(* CODESYS project xlh_ha_00_02.project
   Author: Pascal Helfenstein
   Title: xlh_ha
   Company: xemax ag

Project tree, tasks and I/O mapping:
  xlh_base : CODESYS Control for Raspberry Pi 64 SL, CODESYS, order no. 2302000009, version 4.20.0.0
    application app
      libraries: Standard, 3.5.22.0 (System); StringUtils, 3.5.22.0 (System); VisuDialogs, * (System); Web Socket Client SL, 1.12.0.0 (CODESYS); Net Base Services, * (3S - Smart Software Solutions GmbH); MQTT Client SL, 1.13.0.0 (CODESYS); Util, 3.5.22.0 (System); String Functions, * (CODESYS); SysTimeRtc, * (System); SysTime, 3.5.17.0 (System); CmpIecTask, * (System); Memory, 3.5.17.0 (3S - Smart Software Solutions GmbH)
      task MainTask (cyclic, interval t#20ms, priority 1) calls LOCAL_TIME_AND_TIME_ZONE, TASK_INFO, io, MAIN
      task VISU_TASK (cyclic, interval 100 ms, priority 31) calls VisuElems.Visu_Prg
      program MAIN [ST]
      IoT/
        DEVICES/
          function block _000_FB_VISU_BASE [ST]
          function block _200_FB_DEVICE_SHELLY_BASE [ST]: statusUpdate, startup, newMessage
          function block _202_FB_DEVICE_SHELLY_1PM_TEMP [ST]: newMessage
          interface IDevice
          interface IDeviceZigbee2Mqtt
          interface IDeviceShelly
          function block _201_FB_DEVICE_SHELLY_1PM_PLUG [ST]: publisher, newMessage
          function block _300_FB_DEVICE_Z2M_BASE [ST]: statusUpdate, startup, newMessage
          VISU/
            visualisation VISU_FB_DEVICE_SHELLY_RELAIS
            visualisation VISU_FB_DEVICE_SHELLY_RELAIS_TEMP
            visualisation _310_VISU_FB_DEVICE_Z2M_POWER_SWITCH
            visualisation _311_VISU_FB_DEVICE_Z2M_POWER_SWITCH_IKEAL_INSPELING
            visualisation _312_VISU_FB_DEVICE_Z2M_POWER_LAMP
            visualisation _341_VISU_FB_DEVICE_Z2M_BATTERY_SONOFF_TEMP_HUM
          function block _100_FB_DEVICE [ST]: subscriber, publisher, startup, popFifoPublish, newMessage, statusUpdate, pushFifoPublish
          interface IVisu
          function block _311_FB_DEVICE_Z2M_POWER_SWITCH_IKEA_INSPELING [ST]: newMessage
          function block _312_FB_DEVICE_Z2M_POWER_LAMP [ST]: newMessage, publisher
          function block _310_FB_DEVICE_Z2M_POWER_SWITCH [ST]: statusUpdate, startup, newMessage, publisher
          function block _341_FB_DEVICE_Z2M_BATTERY_SONOFF_TEMP_HUM [ST]: newMessage
          function block _340_FB_DEVICE_Z2M_BATTERY [ST]: newMessage
          function block _342_FB_DEVICE_Z2M_BATTERY_AQARA_SWITCH_H1 [ST]: newMessage
          function block _314_FB_DEVICE_Z2M_SHELLY_EM [ST]: newMessage
          function block _343_FB_DEVICE_Z2M_BATTERY_HUE_SWITCH_DIMMER [ST]: newMessage
          function block _344_FB_DEVICE_Z2M_BATTERY_HUE_MOTION [ST]: newMessage
          function block _345_FB_DEVICE_Z2M_BATTERY_HUE_WALL_SWITCH [ST]: newMessage
          function block _313_FB_DEVICE_Z2M_SHELLY_1PM [ST]: newMessage
        MQTT_Client/
          function TERMINATE_STRING [ST]
          function block FB_MQTT_CLIENT [ST]: pMqttClient, setClientIdNr
          function GET_VALUE_FROM_MSG [ST]
          function GET_REAL_FROM_VALUE [ST]
          function GET_BOOL_FROM_VALUE [ST]
          function GET_INT_FROM_VALUE [ST]
          function GET_STRING_FROM_VALUE [ST]
          function GET_LREAL_FROM_VALUE [ST]
          function GET_BOOL_FROM_VALUE_ON_OFF [ST]
        global variables GC
        program TASK_INFO [ST]
        program LOCAL_TIME_AND_TIME_ZONE [ST]
        FUNCTIONS/
          function block FB_IMPULSE_SWITCH [ST]
      visualisation VISUALIZATION
      io/
        program io [ST]
      program LOGIC [CFC]
    SoftMotion General Axis Pool
    GPIOs_A_B : GPIOs B+/Pi2, CODESYS, version 4.20.0.0
        unmapped channels: digital inputs (GPIO0..GPIO31), digital outputs (GPIO0..GPIO31)
    Onewire
    Camera device
      <Empty>
    SPI
    I²C
  libraries: VisuSymbols, 4.5.0.0 (System)
  text list GlobalTextList
  5ce3da45-db07-42e7-a21c-a00fff4ed8f6|C:\Users\a.werner\Documents\background.jpg
*)

// xlh_base/app/IoT/GC
// =============================================================================
// GC — Global constants (qualified-only)
// -----------------------------------------------------------------------------
// Collects the string sizes used project-wide for MQTT topics and message
// buffers. Changes affect the memory footprint of every device FB.
// =============================================================================
{attribute 'qualified_only'}
VAR_GLOBAL CONSTANT
    STRING_SIZE_TOPIC      : INT := 1024;   // Maximum size of an MQTT topic ((W)STRING length)
    STRING_SIZE_MESSAGE_TX : INT := 1024;   // Maximum size of a transmit message
    STRING_SIZE_MESSAGE_RX : INT := 2048;   // Maximum size of a receive message
END_VAR

// xlh_base/app/IoT/LOCAL_TIME_AND_TIME_ZONE
// =============================================================================
// LOCAL_TIME_AND_TIME_ZONE
// -----------------------------------------------------------------------------
// Provides the current UTC and CET/CEST time and their components
// (year, month, day, hour, ..., weekday, leap year) as program outputs.
//
// Uses the Util library for the time-zone conversion between UTC (RTC)
// and Central European Time (daylight-saving switchover on the last
// Sunday of March/October respectively).
//
// Usage: time-of-day controls (e.g. _344 motion sensor active window).
// =============================================================================
PROGRAM LOCAL_TIME_AND_TIME_ZONE
VAR_OUTPUT
    stUTC_Timestamp      : SysTime;         // RTC timestamp UTC
    stCTE_Timestamp      : SysTime;         // CET/CEST timestamp
    stJoinedTimestamp    : SysTime;         // CET components joined back into a UTC timestamp
    stCombinedTimestamp  : SysTime;         // datDate + todTime combined
    uiYear               : YEAR;            // 1970..2106
    uiMonth              : MONTH;
    uiDay                : DAY;
    uiHour               : UINT;
    uiMinute             : UINT;
    uiSecond             : UINT;
    uiMilliseconds       : MILLISECOND;
    eWeekday             : WEEKDAY;
    datDate              : DATE;
    todTime              : TIME_OF_DAY;
    eError               : Util.ERROR;
    xLeapYear            : BOOL;
END_VAR
VAR CONSTANT
    /// Coordinated Universal Time
    gc_tzTimeZoneUTC : TimeZone := (asgPeriod := [(sName := 'UTC')]);

    /// Central European Time / Central European Summer Time with switchover rules.
    gc_tzTimeZoneCET : TimeZone := (
        iBias := 60 (* T#1M => minutes *),
        asgPeriod := [
            ( (* Summer time -> standard time: last Sunday of October, 03:00 local *)
                sName  := 'CET',
                dtDate := (uiMonth := 10, eWeekday := WEEKDAY.SUNDAY, uiDay := 5, uiHour := 3)
            ),
            ( (* Standard time -> summer time: last Sunday of March, 02:00 local *)
                sName  := 'CEST',
                dtDate := (uiMonth := 3,  eWeekday := WEEKDAY.SUNDAY, uiDay := 5, uiHour := 2),
                iBias  := 60 (* T#1M => minutes *)
            )
        ]
    );
END_VAR

// 1) Read the RTC UTC timestamp.
SysTimeRtcHighResGet(pTimestamp := stUTC_Timestamp);

// 2) UTC -> CET/CEST according to the configured TimeZone.
stCTE_Timestamp := Util.LocalDateTime(tzTimeZone := gc_tzTimeZoneCET,
                                      uliDateTime := stUTC_Timestamp,
                                      eErrorID    => eError);

// 3) Split the CET timestamp into its individual components.
eError := Util.SplitDateTime(uliDateTime    := stCTE_Timestamp,
                             uiYear         => uiYear,
                             uiMonth        => uiMonth,
                             uiDay          => uiDay,
                             uiHour         => uiHour,
                             uiMinute       => uiMinute,
                             uiSecond       => uiSecond,
                             uiMilliseconds => uiMilliseconds,
                             eWeekday       => eWeekday);

// 4) Join the components back into a UTC timestamp (diagnostics).
stJoinedTimestamp := Util.JoinDateTime(uiYear         := uiYear,
                                       uiMonth        := uiMonth,
                                       uiDay          := uiDay,
                                       uiHour         := uiHour,
                                       uiMinute       := uiMinute,
                                       uiSecond       := uiSecond,
                                       uiMilliseconds := uiMilliseconds);

// 5) Derive the IEC-typed parts (datDate, todTime).
Util.SeparateDateTime(uliDateTime := stCTE_Timestamp,
                      eWeekDay    => eWeekDay,
                      datDate     => datDate,
                      todTime     => todTime);

// 6) Reconstruct a timestamp from datDate + todTime.
stCombinedTimestamp := Util.CombineDateTime(datDate  := datDate,
                                            todTime  := todTime,
                                            eErrorID => eError);

// 7) Calculate the weekday from the date (verification).
eWeekday := Util.DayOfWeek(datDate := datDate, eErrorID => eError);

// 8) Leap-year flag.
xLeapYear := Util.IsLeapYear(uiYear := uiYear, eErrorID => eError);

END_PROGRAM

// xlh_base/app/IoT/TASK_INFO
// =============================================================================
// TASK_INFO
// -----------------------------------------------------------------------------
// Reads the key figures of the current task (interval, jitter, effective
// cycle time) at runtime via the CmpIecTask library and makes them available
// to all POUs through program outputs.
//
// Usage in the device FBs: integration of energy via fCycleTime, periodic
// status queries via fCycleTime-based second counters.
//
// Sources:
//   https://content.helpme-codesys.com/en/libs/CmpIecTask/Current/index.html
//   https://forge.codesys.com/forge/talk/Engineering/thread/b7e9b2b353/
//   https://medium.com/@sean.gongz/...how-to-get-current-task-actual-cycle-time-in-codesys
// =============================================================================
PROGRAM TASK_INFO
VAR
    Result            : CmpIecTask.RTS_IEC_RESULT;
    hCurrentTask      : CmpIecTask.RTS_IEC_HANDLE;
    pCurrentTaskInfo  : POINTER TO Task_Info2;
    stCurrentTaskInfo : Task_Info2;
END_VAR
VAR_OUTPUT
    fCycleTime              : LREAL;    // Effective cycle time in seconds (interval + jitter)
    fInterval               : LREAL;    // Configured task interval (us)
    fCycleTimeUs            : LREAL;    // Effective cycle time in microseconds
    fJitterUs               : LREAL;    // Current jitter (us)
    fJitterOffsetInterwalUs : LREAL;    // Interval + jitter (us)
END_VAR

// Get the current task handle and dereference the info structure.
hCurrentTask      := IecTaskGetCurrent(pResult := ADR(Result));
pCurrentTaskInfo  := IecTaskGetInfo3(hIecTask := hCurrentTask, pResult := ADR(Result));
stCurrentTaskInfo := pCurrentTaskInfo^;

// Prepare the results.
fCycleTimeUs            := TO_LREAL(TO_DINT(stCurrentTaskInfo.dwInterval) + stCurrentTaskInfo.iJitter);
fInterval               := TO_LREAL(stCurrentTaskInfo.dwInterval);
fJitterUs               := TO_LREAL(stCurrentTaskInfo.iJitter);
fJitterOffsetInterwalUs := fInterval + fJitterUs;
fCycleTime              := fCycleTimeUs / 1000000.0;

END_PROGRAM

// xlh_base/app/io/io
// =============================================================================
// io
// -----------------------------------------------------------------------------
// Central device program: instantiates all devices connected via
// Zigbee2MQTT/Shelly (as VAR_INPUT so they can be parameterized via the
// visualization / online), binds them to shared FB_MQTT_CLIENT instances
// and calls them cyclically.
//
// Architecture:
//   - Devices are not assigned directly to one MQTT client but are managed
//     through a pointer array (_aIoClients).
//   - Several FB_MQTT_CLIENT instances (_afbMqttClient) are used so that
//     the MQTT library is not overloaded by too many parallel subscribes.
//     iNR_OF_IO_TO_ONE_MQTT_CLIENT devices are bundled per MQTT client.
//   - The initial configuration (pointer binding, topics) is done once in
//     the startup block.
// =============================================================================
PROGRAM io
VAR_INPUT
    // Zigbee wireless switches / sensors (battery devices)
    fbSwitch1       : _343_FB_DEVICE_Z2M_BATTERY_HUE_SWITCH_DIMMER := (bEnable:=TRUE, sMqttTopicBase:='switch_1', sLabel:='');
    fbSwitch2       : _345_FB_DEVICE_Z2M_BATTERY_HUE_WALL_SWITCH   := (bEnable:=TRUE, sMqttTopicBase:='switch_2', sLabel:='');
    fbTempHumSensor : _341_FB_DEVICE_Z2M_BATTERY_SONOFF_TEMP_HUM   := (bEnable:=TRUE, sMqttTopicBase:='temp_hum_sensor', sLabel:='');
    fbMotionSensor: _344_FB_DEVICE_Z2M_BATTERY_HUE_MOTION       := (bEnable:=TRUE, sMqttTopicBase:='motion_sensor', sLabel:='');

    // Zigbee switch actuators / lamps / energy meters
    fbLamp1   : _312_FB_DEVICE_Z2M_POWER_LAMP                       := (bEnable:=TRUE, sMqttTopicBase:='lamp_1',  sLabel:='');
    fbLamp2   : _312_FB_DEVICE_Z2M_POWER_LAMP                       := (bEnable:=TRUE, sMqttTopicBase:='lamp_2',  sLabel:='');
    fbPlug1   : _310_FB_DEVICE_Z2M_POWER_SWITCH                     := (bEnable:=TRUE, sMqttTopicBase:='plug_1',  sLabel:='');
    fbPlug2   : _311_FB_DEVICE_Z2M_POWER_SWITCH_IKEA_INSPELING      := (bEnable:=TRUE, sMqttTopicBase:='plug_2',  sLabel:='');
    fbShelly1 : _313_FB_DEVICE_Z2M_SHELLY_1PM                       := (bEnable:=TRUE, sMqttTopicBase:='shelly_1', sLabel:='');
    fbShelly2 : _314_FB_DEVICE_Z2M_SHELLY_EM                        := (bEnable:=TRUE, sMqttTopicBase:='shelly_2', sLabel:='');
END_VAR
VAR CONSTANT
    iNR_OF_IO_CLIENTS            : INT := 100; // Maximum number of devices in the pointer array
    iNR_OF_MQTT_CLIENTS          : INT :=  20; // Number of MQTT clients (connections to the broker)
    iNR_OF_IO_TO_ONE_MQTT_CLIENT : INT :=   5; // Devices per MQTT client
END_VAR
VAR
    _bStartup     : BOOL := TRUE;                                                     // One-time initialization
    _aIoClients   : ARRAY[0..(iNR_OF_IO_CLIENTS   - 1)] OF POINTER TO _100_FB_DEVICE; // Device pointer array
    _afbMqttClient: ARRAY[0..(iNR_OF_MQTT_CLIENTS - 1)] OF FB_MQTT_CLIENT;            // Distributed MQTT clients
    _iI           : INT;
    _iN           : INT;
END_VAR

// =============================================================================
// One-time initialization
// -----------------------------------------------------------------------------
// 1. Register the devices in the pointer array (the order determines the
//    assignment to the MQTT clients).
// 2. Set the ClientId per MQTT client (xlh_base_ha_io_<n>).
// 3. Bind the devices to their MQTT client pointer and call startup().
// 4. Enable the MQTT clients (bEnable := TRUE).
// =============================================================================
IF _bStartup THEN
    _bStartup := FALSE;

    // (1) Register the devices.
    _iI := 0;
    _aIoClients[_iI] := ADR(fbSwitch1);       _iI := _iI + 1;
    _aIoClients[_iI] := ADR(fbSwitch2);       _iI := _iI + 1;
    _aIoClients[_iI] := ADR(fbTempHumSensor); _iI := _iI + 1;
    _aIoClients[_iI] := ADR(fbMotionSensor);  _iI := _iI + 1;

    _aIoClients[_iI] := ADR(fbLamp1);         _iI := _iI + 1;
    _aIoClients[_iI] := ADR(fbLamp2);         _iI := _iI + 1;
    _aIoClients[_iI] := ADR(fbPlug1);         _iI := _iI + 1;
    _aIoClients[_iI] := ADR(fbPlug2);         _iI := _iI + 1;
    _aIoClients[_iI] := ADR(fbShelly1);       _iI := _iI + 1;
    _aIoClients[_iI] := ADR(fbShelly2);       _iI := _iI + 1;

    // (2) Set unique client ids.
    FOR _iI := 0 TO (iNR_OF_MQTT_CLIENTS - 1) BY 1 DO
        _afbMqttClient[_iI].setClientIdNr(sClientId := 'xlh_base_ha_io_', iNr := _iI);
    END_FOR

    // (3) Bind the devices to the MQTT clients and initialize them.
    FOR _iI := 0 TO (iNR_OF_IO_CLIENTS - 1) BY 1 DO
        IF _aIoClients[_iI] > 16#0 THEN
            _iN := _iI / iNR_OF_IO_TO_ONE_MQTT_CLIENT;
            _aIoClients[_iI]^.pMqttClient := ADR(_afbMqttClient[_iN]);
            _aIoClients[_iI]^.startup();
        END_IF
    END_FOR

    // (4) Enable the MQTT clients.
    FOR _iI := 0 TO (iNR_OF_MQTT_CLIENTS - 1) BY 1 DO
        _afbMqttClient[_iI].bEnable := TRUE;
    END_FOR
END_IF

// =============================================================================
// Cyclic calls
// =============================================================================
// MQTT clients first -> required so the subscribers/publishers of the
// devices see an up-to-date connection state.
FOR _iI := 0 TO (iNR_OF_MQTT_CLIENTS - 1) BY 1 DO
    _afbMqttClient[_iI]();
END_FOR

// Call the devices.
FOR _iI := 0 TO (iNR_OF_IO_CLIENTS - 1) BY 1 DO
    IF _aIoClients[_iI] > 16#0 THEN
        _aIoClients[_iI]^();
    END_IF
END_FOR

END_PROGRAM

// xlh_base/app/IoT/MQTT_Client/FB_MQTT_CLIENT
// =============================================================================
// FB_MQTT_CLIENT
// -----------------------------------------------------------------------------
// Wrapper around the IoTCommonLib MQTT.MQTTClient. Provides a simplified
// interface (Enable / Hostname / ClientId) and returns the connection and
// error status flags.
//
// Properties / methods:
//   - pMqttClient    : Property GET, returns a pointer to the internal MQTT
//                      client (used by device FBs to bind their own
//                      subscribe/publish blocks to the client).
//   - setClientIdNr  : Helper method to create a unique client id by
//                      appending a sequential number.
// =============================================================================
FUNCTION_BLOCK FB_MQTT_CLIENT
VAR_INPUT
    bEnable   : BOOL;                       // TRUE = activate the connection
    sHostname : STRING(255) := 'localhost'; // Hostname of the MQTT broker
    sClientId : STRING(255) := 'xLH_mqtt_codesys'; // Unique client id
END_VAR
VAR_OUTPUT
    bConnected  : BOOL;                     // TRUE = connected to the broker
    bError      : BOOL;                     // TRUE = connection/protocol error
    fbMqttClient: MQTT.MQTTClient := (
        uiPort             := 1883,
        eMQTTVersion       := MQTT.MQTT_VERSION.V3_1_1,
        eCommunicationMode := MQTT.COMMUNICATION_MODE.TCP); // Internal client (referenced by pMqttClient)
END_VAR

// Control the MQTT client: while the error flag is active, xEnable is
// automatically reset so the IoTCommon library can reset internally.
fbMqttClient.xEnable   := bEnable AND NOT fbMqttClient.xError;
fbMqttClient.sClientId := sClientId;
fbMqttClient(sHostname := sHostname);

// Status outputs.
bConnected := fbMqttClient.xConnectedToBroker;
bError     := fbMqttClient.xError;

// =============================================================================
// PROPERTY pMqttClient (GET)
// -----------------------------------------------------------------------------
// Returns a pointer to the internal MQTT client so that device FBs can
// couple their MQTT.MQTTSubscribe / MQTT.MQTTPublish instances to the same
// connection.
// =============================================================================
PROPERTY pMqttClient : POINTER TO FB_MQTT_CLIENT
GET
pMqttClient := ADR(THIS^.fbMqttClient);
END_GET
END_PROPERTY

// =============================================================================
// METHOD setClientIdNr
// -----------------------------------------------------------------------------
// Sets the client id by appending a sequential number to a base name.
// Used by the io program to create a unique id per MQTT client instance
// ('xlh_base_ha_io_0', '..._1', ...).
// =============================================================================
METHOD setClientIdNr : BOOL
VAR_INPUT
    sClientId : STRING(255) := 'xLH_mqtt_codesys'; // Base id
    iNr       : INT;                                // Number to append
END_VAR
VAR
    sNumber : STRING(255);
END_VAR
sNumber := TO_STRING(iNr);
THIS^.sClientId := CONCAT(sClientId, sNumber);
END_METHOD

END_FUNCTION_BLOCK

// xlh_base/app/IoT/DEVICES/_343_FB_DEVICE_Z2M_BATTERY_HUE_SWITCH_DIMMER
// =============================================================================
// _343_FB_DEVICE_Z2M_BATTERY_HUE_SWITCH_DIMMER
// -----------------------------------------------------------------------------
// Philips Hue Dimmer Switch (4 buttons: On / Off / Up / Down) with
// press / hold / release actions per button.
// Device link: https://www.zigbee2mqtt.io/devices/929002398602.html
//
// Behavior of the boolean outputs:
//   - Pulses: set for EXACTLY ONE PLC cycle when an action is received,
//     reset again in the following cycle.
// =============================================================================
FUNCTION_BLOCK _343_FB_DEVICE_Z2M_BATTERY_HUE_SWITCH_DIMMER EXTENDS _340_FB_DEVICE_Z2M_BATTERY
VAR_OUTPUT
    sAction          : STRING(255);   // Last reported action (diagnostics)

    // ON button
    bOnPress         : BOOL;
    bOnPressRelease  : BOOL;
    bOnHold          : BOOL;
    bOnHoldRelease   : BOOL;

    // OFF button
    bOffPress        : BOOL;
    bOffPressRelease : BOOL;
    bOffHold         : BOOL;
    bOffHoldRelease  : BOOL;

    // UP button
    bUpPress         : BOOL;
    bUpPressRelease  : BOOL;
    bUpHold          : BOOL;
    bUpHoldRelease   : BOOL;

    // DOWN button
    bDownPress       : BOOL;
    bDownPressRelease: BOOL;
    bDownHold        : BOOL;
    bDownHoldRelease : BOOL;
END_VAR
VAR
    _bNewAction : BOOL;
END_VAR

SUPER^();

IF _bNewAction THEN
    _bNewAction := FALSE;

    bOnPress          := sAction = 'on_press';
    bOnPressRelease   := sAction = 'on_press_release';
    bOnHold           := sAction = 'on_hold';
    bOnHoldRelease    := sAction = 'on_hold_release';

    bOffPress         := sAction = 'off_press';
    bOffPressRelease  := sAction = 'off_press_release';
    bOffHold          := sAction = 'off_hold';
    bOffHoldRelease   := sAction = 'off_hold_release';

    bUpPress          := sAction = 'up_press';
    bUpPressRelease   := sAction = 'up_press_release';
    bUpHold           := sAction = 'up_hold';
    bUpHoldRelease    := sAction = 'up_hold_release';

    bDownPress        := sAction = 'down_press';
    bDownPressRelease := sAction = 'down_press_release';
    bDownHold         := sAction = 'down_hold';
    bDownHoldRelease  := sAction = 'down_hold_release';
ELSE
    bOnPress          := FALSE;
    bOnPressRelease   := FALSE;
    bOnHold           := FALSE;
    bOnHoldRelease    := FALSE;

    bOffPress         := FALSE;
    bOffPressRelease  := FALSE;
    bOffHold          := FALSE;
    bOffHoldRelease   := FALSE;

    bUpPress          := FALSE;
    bUpPressRelease   := FALSE;
    bUpHold           := FALSE;
    bUpHoldRelease    := FALSE;

    bDownPress        := FALSE;
    bDownPressRelease := FALSE;
    bDownHold         := FALSE;
    bDownHoldRelease  := FALSE;
END_IF

// =============================================================================
// METHOD newMessage
// -----------------------------------------------------------------------------
// Reads the action from the event topic and triggers the pulse logic in
// the next cycle.
// =============================================================================
METHOD newMessage : BOOL
SUPER^.newMessage();
IF _fbMqttSubscriber.wsLastTopic = _wsMqttTopicEvent THEN
    sAction := GET_STRING_FROM_VALUE(sAction, GET_VALUE_FROM_MSG('action', ADR(_sSubscribedMessage)));
    THIS^._bNewAction := TRUE;
END_IF
END_METHOD

END_FUNCTION_BLOCK

// xlh_base/app/IoT/DEVICES/_340_FB_DEVICE_Z2M_BATTERY
// =============================================================================
// _340_FB_DEVICE_Z2M_BATTERY
// -----------------------------------------------------------------------------
// Base FB for battery-powered Zigbee devices. Reads the battery level
// (battery, 0..100%) from the Z2M event topic.
//
// Derived by sensors (_341, _344) and push buttons/switches (_342, _343,
// _345).
// =============================================================================
FUNCTION_BLOCK _340_FB_DEVICE_Z2M_BATTERY EXTENDS _300_FB_DEVICE_Z2M_BASE
VAR_OUTPUT
    iBattery : INT := -1;       // Battery level 0..100% (-1 = unknown)
END_VAR

SUPER^();

// =============================================================================
// METHOD newMessage
// -----------------------------------------------------------------------------
// Reads the battery level from the Z2M event topic.
// =============================================================================
METHOD newMessage : BOOL
SUPER^.newMessage();
IF _fbMqttSubscriber.wsLastTopic = _wsMqttTopicEvent THEN
    iBattery := GET_INT_FROM_VALUE(iBattery, GET_VALUE_FROM_MSG('battery', ADR(_sSubscribedMessage)));
END_IF
END_METHOD

END_FUNCTION_BLOCK

// xlh_base/app/IoT/DEVICES/_300_FB_DEVICE_Z2M_BASE
// =============================================================================
// _300_FB_DEVICE_Z2M_BASE
// -----------------------------------------------------------------------------
// Base FB for Zigbee2MQTT devices. Provides the standard Z2M topics and
// parses the common 'linkquality' field.
//
// Standard topic schema (Zigbee2MQTT):
//   zigbee2mqtt/<base>          (subscribe filter via wildcard ".../#")
//   zigbee2mqtt/<base>          -> event topic (status pushes from the device)
//   zigbee2mqtt/<base>/set      -> publish: action to the device
//   zigbee2mqtt/<base>/get      -> publish: trigger a status query
//
// Example:
//   Set output
//     zigbee2mqtt/plug_1/set    {"state": "OFF"} | {"state": "ON"}
//   Status query
//     zigbee2mqtt/plug_1/get    {"state":""}
// =============================================================================
FUNCTION_BLOCK _300_FB_DEVICE_Z2M_BASE EXTENDS _100_FB_DEVICE IMPLEMENTS IDeviceZigbee2Mqtt
VAR_INPUT
    sMqttTopicZigbee2Mqtt : STRING(255) := 'zigbee2mqtt';   // Z2M prefix (usually 'zigbee2mqtt')
END_VAR
VAR_OUTPUT
    iLinkquality : INT := -1;       // Zigbee link quality (-1 = unknown)
END_VAR
VAR
    _wsMqttTopicZigbee2Mqtt : WSTRING(GC.STRING_SIZE_TOPIC); // sMqttTopicZigbee2Mqtt as WSTRING
    _wsMqttTopicEvent       : WSTRING(GC.STRING_SIZE_TOPIC); // zigbee2mqtt/<base>
    _wsMqttTopicSet         : WSTRING(GC.STRING_SIZE_TOPIC); // zigbee2mqtt/<base>/set
    _wsMqttTopicGet         : WSTRING(GC.STRING_SIZE_TOPIC); // zigbee2mqtt/<base>/get
END_VAR

SUPER^();

// =============================================================================
// METHOD statusUpdate
// -----------------------------------------------------------------------------
// Hook (no own code) — overridden by derived FBs.
// =============================================================================
METHOD statusUpdate : BOOL
SUPER^.statusUpdate();
END_METHOD

// =============================================================================
// METHOD startup
// -----------------------------------------------------------------------------
// Builds the subscribe filter and all Z2M-specific topic strings.
// =============================================================================
METHOD startup : BOOL
SUPER^.startup();
THIS^._wsMqttTopicZigbee2Mqtt := STRING_TO_WSTRING(sMqttTopicZigbee2Mqtt);

// Subscribe filter: zigbee2mqtt/<base>/#
_wsSubcribedTopicFilter := "";
Stu.StrConcatW(pstFrom:=ADR(THIS^._wsMqttTopicZigbee2Mqtt), pstTo:=ADR(_wsSubcribedTopicFilter), iBufferSize:=GC.STRING_SIZE_TOPIC);
Stu.StrConcatW(pstFrom:=ADR("/"),                          pstTo:=ADR(_wsSubcribedTopicFilter), iBufferSize:=GC.STRING_SIZE_TOPIC);
Stu.StrConcatW(pstFrom:=ADR(THIS^._wsMqttTopicBase),       pstTo:=ADR(_wsSubcribedTopicFilter), iBufferSize:=GC.STRING_SIZE_TOPIC);
Stu.StrConcatW(pstFrom:=ADR("/#"),                         pstTo:=ADR(_wsSubcribedTopicFilter), iBufferSize:=GC.STRING_SIZE_TOPIC);

// Event topic: zigbee2mqtt/<base>
_wsMqttTopicEvent := "";
Stu.StrConcatW(pstFrom:=ADR(THIS^._wsMqttTopicZigbee2Mqtt), pstTo:=ADR(_wsMqttTopicEvent), iBufferSize:=GC.STRING_SIZE_TOPIC);
Stu.StrConcatW(pstFrom:=ADR("/"),                          pstTo:=ADR(_wsMqttTopicEvent), iBufferSize:=GC.STRING_SIZE_TOPIC);
Stu.StrConcatW(pstFrom:=ADR(THIS^._wsMqttTopicBase),       pstTo:=ADR(_wsMqttTopicEvent), iBufferSize:=GC.STRING_SIZE_TOPIC);

// Set topic: zigbee2mqtt/<base>/set
_wsMqttTopicSet := "";
Stu.StrConcatW(pstFrom:=ADR(_wsMqttTopicEvent), pstTo:=ADR(_wsMqttTopicSet), iBufferSize:=GC.STRING_SIZE_TOPIC);
Stu.StrConcatW(pstFrom:=ADR("/set"),            pstTo:=ADR(_wsMqttTopicSet), iBufferSize:=GC.STRING_SIZE_TOPIC);

// Get topic: zigbee2mqtt/<base>/get
_wsMqttTopicGet := "";
Stu.StrConcatW(pstFrom:=ADR(_wsMqttTopicEvent), pstTo:=ADR(_wsMqttTopicGet), iBufferSize:=GC.STRING_SIZE_TOPIC);
Stu.StrConcatW(pstFrom:=ADR("/get"),            pstTo:=ADR(_wsMqttTopicGet), iBufferSize:=GC.STRING_SIZE_TOPIC);
END_METHOD

// =============================================================================
// METHOD newMessage
// -----------------------------------------------------------------------------
// Reads the link quality (available for all Z2M devices) from the event
// topic.
// =============================================================================
METHOD newMessage : BOOL
SUPER^.newMessage();
IF _fbMqttSubscriber.wsLastTopic = _wsMqttTopicEvent THEN
    iLinkquality := GET_INT_FROM_VALUE(iLinkquality, GET_VALUE_FROM_MSG('linkquality', ADR(_sSubscribedMessage)));
END_IF
END_METHOD

END_FUNCTION_BLOCK

// xlh_base/app/IoT/DEVICES/_100_FB_DEVICE
// =============================================================================
// _100_FB_DEVICE
// -----------------------------------------------------------------------------
// Generic MQTT device base class. Connects one MQTT subscriber and one MQTT
// publisher instance to an externally referenced FB_MQTT_CLIENT and provides
// a publish queue (LIFO).
//
// Usage:
//   1. Externally assign pMqttClient (pointer to FB_MQTT_CLIENT) and
//      sMqttTopicBase in the calling program.
//   2. Call the method startup() once for commissioning (the topic filters
//      are built).
//   3. bEnable := TRUE -> the subscriber subscribes to sMqttTopicBase + '/#'
//      and calls newMessage() for every message.
//
// Extension in derived FBs:
//   - newMessage()    : Parse the message and update the outputs.
//   - publisher()     : Enqueue MQTT messages via pushFifoPublish().
//   - statusUpdate()  : Called once on every subscribe re-/connect
//                       (e.g. to send active status queries).
//
// Publish queue:
//   The methods push/popFifoPublish implement a LIFO with a fixed depth of
//   _iFIFO_SIZE. An internal cycle-delay counter prevents several publishes
//   from following each other without a pause (relieves the broker and the
//   MQTT library).
// =============================================================================
FUNCTION_BLOCK _100_FB_DEVICE EXTENDS _000_FB_VISU_BASE IMPLEMENTS IDevice
VAR_INPUT
    bEnable        : BOOL;                          // TRUE -> subscriber/publisher active
    sMqttTopicBase : STRING(255);                   // Base topic of the device (without wildcard)
    pMqttClient    : POINTER TO FB_MQTT_CLIENT;     // Pointer to the shared MQTT client
END_VAR
VAR
    // ---- Topic strings (caches) -----------------------------------------------
    _wsMqttTopicBase         : WSTRING(GC.STRING_SIZE_TOPIC); // sMqttTopicBase as WSTRING
    _wsSubcribedTopicFilter  : WSTRING(GC.STRING_SIZE_TOPIC); // _wsMqttTopicBase + '/#'

    // ---- Connection triggers and watchdogs ------------------------------------
    _fbRtMqttClientConnected : R_TRIG;                // Rising edge:  MQTT connection established
    _fbFtMqttClientConnected : F_TRIG;                // Falling edge: MQTT connection lost
    _fbRtMqttSubscriberActive: R_TRIG;                // Subscriber became active (-> statusUpdate)
    _fbFtMqttSubscriberActive: F_TRIG;
    _fbRtError               : R_TRIG;                // Error edge of the MQTT client
    _fbTonConnect            : TON;                   // Reconnect delay (subscribe enable)
    _fbTonDisconnect         : TON;                   // Watchdog (subscribe disable when stale)

    // ---- Subscriber -----------------------------------------------------------
    _fbMqttSubscriber : MQTT.MQTTSubscribe;
    _sSubscribedMessage : STRING(GC.STRING_SIZE_MESSAGE_RX);

    // ---- Publisher (current slot) ---------------------------------------------
    _fbMqttPublisher : MQTT.MQTTPublish;
    _wsPublishTopic  : WSTRING(GC.STRING_SIZE_TOPIC);
    _sPublishMessage : STRING(GC.STRING_SIZE_MESSAGE_TX);

    // ---- Publisher queue (LIFO) -----------------------------------------------
    _iFifoPos             : INT;       // Current fill level
    _iFifoPosMax          : INT;       // Maximum value (watermark) for diagnostics
    _iFifoPopCycleCounter : INT;       // Cycle delay between pop operations
    _awsPublishTopic   : ARRAY[0..(_iFIFO_SIZE - 1)] OF WSTRING(GC.STRING_SIZE_TOPIC);
    _asPublishMessage  : ARRAY[0..(_iFIFO_SIZE - 1)] OF STRING(GC.STRING_SIZE_MESSAGE_TX);

    // ---- Diagnostics ----------------------------------------------------------
    _todMessageUpdate : TIME_OF_DAY;   // Time of day of the last received message
END_VAR
VAR CONSTANT
    _iFIFO_SIZE          : INT := 30; // Depth of the publish queue
    _iFIFO_DELAY_COUNTER : INT := 5;  // Cycles of pause between two publish pop operations
END_VAR

THIS^.subscriber();
THIS^.publisher();

// =============================================================================
// METHOD subscriber
// -----------------------------------------------------------------------------
// Manages the life cycle of the MQTT subscriber and calls newMessage() for
// new messages and statusUpdate() on (re-)activation.
//
// Logic:
//   - The subscriber is activated when the connection is established and
//     deactivated on disconnect / error.
//   - Watchdog _fbTonDisconnect (3s): if the subscriber is enabled but not
//     busy, it is briefly disabled to reset the library.
//   - After _fbTonConnect (500ms) the subscriber is activated again.
// =============================================================================
METHOD subscriber : BOOL
THIS^._fbRtMqttClientConnected(CLK := THIS^.pMqttClient^.bConnected);
THIS^._fbFtMqttClientConnected(CLK := THIS^.pMqttClient^.bConnected);
THIS^._fbRtError              (CLK := THIS^.pMqttClient^.bError);

// Activate the subscriber on connect, deactivate it on error/disconnect.
IF THIS^._fbRtMqttClientConnected.Q THEN
    THIS^._fbMqttSubscriber.xEnable := TRUE;
END_IF
IF THIS^._fbRtError.Q OR THIS^._fbFtMqttClientConnected.Q THEN
    THIS^._fbMqttSubscriber.xEnable := FALSE;
END_IF

// Watchdog: stalled subscriber -> brief reset.
THIS^._fbTonDisconnect.IN := THIS^.pMqttClient^.bConnected
                              AND THIS^._fbMqttSubscriber.xEnable
                              AND NOT THIS^._fbMqttSubscriber.xBusy;
THIS^._fbTonDisconnect(PT := T#3000MS);
IF THIS^._fbTonDisconnect.Q THEN
    THIS^._fbMqttSubscriber.xEnable := FALSE;
END_IF

// Reconnect delay.
THIS^._fbTonConnect.IN := THIS^.pMqttClient^.bConnected AND NOT THIS^._fbMqttSubscriber.xEnable;
THIS^._fbTonConnect(PT := T#500MS);
IF THIS^._fbTonConnect.Q THEN
    THIS^._fbMqttSubscriber.xEnable := TRUE;
END_IF

// Device itself disabled -> subscriber off.
IF NOT THIS^.bEnable THEN
    THIS^._fbMqttSubscriber.xEnable := FALSE;
END_IF

// Call the subscriber and null-terminate the received message.
THIS^._fbMqttSubscriber(mqttClient        := THIS^.pMqttClient^.fbMqttClient,
                        wsTopicFilter     := THIS^._wsSubcribedTopicFilter,
                        pbPayload         := ADR(THIS^._sSubscribedMessage),
                        udiMaxPayloadSize := SIZEOF(THIS^._sSubscribedMessage));
TERMINATE_STRING(psIn := ADR(THIS^._sSubscribedMessage), udiLength := THIS^._fbMqttSubscriber.udiPayloadSize);

// On a new message, branch into the derived processing.
IF THIS^._fbMqttSubscriber.xReceived THEN
    THIS^.newMessage();
END_IF

// React to subscriber activation -> status initialization.
THIS^._fbRtMqttSubscriberActive(CLK := THIS^._fbMqttSubscriber.xSubscribeActive);
THIS^._fbFtMqttSubscriberActive(CLK := THIS^._fbMqttSubscriber.xSubscribeActive);
IF THIS^._fbRtMqttSubscriberActive.Q THEN
    THIS^.statusUpdate();
END_IF

// Make values visible for online trace / watch.
_bDummy  := THIS^._fbMqttSubscriber.xEnable;
_bDummy  := THIS^._fbMqttSubscriber.xDone;
_bDummy  := THIS^._fbMqttSubscriber.xBusy;
_bDummy  := THIS^._fbMqttSubscriber.xError;
_bDummy  := THIS^._fbMqttSubscriber.xSubscribeActive;
_wsDummy := THIS^._fbMqttSubscriber.wsLastTopic;
_sDummy  := THIS^._sSubscribedMessage;
END_METHOD

// =============================================================================
// METHOD publisher
// -----------------------------------------------------------------------------
// Controls the MQTT publisher instance: fetches the next message from the
// queue (popFifoPublish), starts the publish and triggers the next
// processing as soon as the current action has finished.
// =============================================================================
METHOD publisher : BOOL
IF THIS^.bEnable THEN
    IF NOT THIS^._fbMqttPublisher.xExecute AND NOT THIS^._fbMqttPublisher.xBusy THEN
        THIS^._fbMqttPublisher.xExecute := popFifoPublish();
    END_IF
ELSE
    THIS^._fbMqttPublisher.xExecute := FALSE;
END_IF

THIS^._fbMqttPublisher(mqttClient     := THIS^.pMqttClient^.fbMqttClient,
                       wsTopicName    := _wsPublishTopic,
                       udiTimeOut     := 10000,
                       pbPayload      := ADR(_sPublishMessage),
                       udiPayloadSize := DINT_TO_UDINT(Stu.StrLenA(ADR(_sPublishMessage))));

IF NOT THIS^._fbMqttPublisher.xBusy OR THIS^._fbMqttPublisher.xError THEN
    THIS^._fbMqttPublisher.xExecute := FALSE;
END_IF
END_METHOD

// =============================================================================
// METHOD startup
// -----------------------------------------------------------------------------
// Initializes the topic strings. Must be called once after sMqttTopicBase
// has been configured (see the io program).
// =============================================================================
METHOD startup : BOOL
VAR_INPUT
END_VAR
_wsMqttTopicBase := STRING_TO_WSTRING(sMqttTopicBase);

// Subscribe filter: <base>/# (all subtopics).
_wsSubcribedTopicFilter := "";
Stu.StrConcatW(pstFrom:=ADR(_wsMqttTopicBase), pstTo:=ADR(_wsSubcribedTopicFilter), iBufferSize:=GC.STRING_SIZE_TOPIC);
Stu.StrConcatW(pstFrom:=ADR("/#"),             pstTo:=ADR(_wsSubcribedTopicFilter), iBufferSize:=GC.STRING_SIZE_TOPIC);
END_METHOD

// =============================================================================
// METHOD popFifoPublish
// -----------------------------------------------------------------------------
// Fetches the next message from the queue (position 0) into the active
// publish slot (_wsPublishTopic / _sPublishMessage). Between two pop
// operations, a pause of _iFIFO_DELAY_COUNTER cycles is made.
// Returns: TRUE if an entry was taken over.
// =============================================================================
METHOD popFifoPublish : BOOL
VAR
    iI : INT;
END_VAR
IF _iFifoPos > 0 AND _iFifoPopCycleCounter = 0 THEN
    _iFifoPos := _iFifoPos - 1;

    // Transfer the message to publish from slot 0 into the publish slot.
    MEM.MemMove(ADR(_awsPublishTopic[0]),  ADR(_wsPublishTopic),  SIZEOF(_wsPublishTopic));
    MEM.MemMove(ADR(_asPublishMessage[0]), ADR(_sPublishMessage), SIZEOF(_sPublishMessage));

    // Shift the remaining entries forward by one position.
    FOR iI := 1 TO (_iFIFO_SIZE - 1) BY 1 DO
        MEM.MemMove(ADR(_awsPublishTopic[iI]),  ADR(_awsPublishTopic[iI - 1]),  SIZEOF(_awsPublishTopic[iI - 1]));
        MEM.MemMove(ADR(_asPublishMessage[iI]), ADR(_asPublishMessage[iI - 1]), SIZEOF(_asPublishMessage[iI - 1]));
    END_FOR

    // Clear the last slot.
    MEM.MemFill(ADR(_awsPublishTopic[_iFIFO_SIZE - 1]),  SIZEOF(_awsPublishTopic[_iFIFO_SIZE - 1]),  16#00);
    MEM.MemFill(ADR(_asPublishMessage[_iFIFO_SIZE - 1]), SIZEOF(_asPublishMessage[_iFIFO_SIZE - 1]), 16#00);

    _iFifoPopCycleCounter := _iFIFO_DELAY_COUNTER;
    popFifoPublish := TRUE;
ELSE
    IF _iFifoPopCycleCounter > 0 THEN
        _iFifoPopCycleCounter := _iFifoPopCycleCounter - 1;
    END_IF
    popFifoPublish := FALSE;
END_IF
END_METHOD

// =============================================================================
// METHOD newMessage
// -----------------------------------------------------------------------------
// Hook for derived FBs: called for every newly received MQTT message.
// Here it only stores the receive time for diagnostic purposes.
// =============================================================================
METHOD newMessage : BOOL
THIS^._todMessageUpdate := LOCAL_TIME_AND_TIME_ZONE.todTime;
END_METHOD

// =============================================================================
// METHOD statusUpdate
// -----------------------------------------------------------------------------
// Hook for derived FBs: called on (re-)activation of the subscriber —
// typical use: send an active status query to the device.
// =============================================================================
METHOD statusUpdate : BOOL
END_METHOD

// =============================================================================
// METHOD pushFifoPublish
// -----------------------------------------------------------------------------
// Puts an MQTT message into the publish queue (at position 0). Existing
// entries are shifted back by one position.
// The call is non-blocking; if the queue is full, FALSE is returned and
// the message is discarded.
// =============================================================================
METHOD pushFifoPublish : BOOL
VAR_INPUT
    wsTopic  : WSTRING(GC.STRING_SIZE_TOPIC);
    sMessage : STRING(GC.STRING_SIZE_MESSAGE_TX);
END_VAR
VAR
    iI : INT;
END_VAR
IF THIS^.bEnable AND _iFifoPos < (_iFIFO_SIZE - 1) THEN
    _iFifoPos := _iFifoPos + 1;

    // Shift the existing entries back by one position (index 0 becomes free).
    FOR iI := (_iFIFO_SIZE - 2) TO 0 BY -1 DO
        MEM.MemMove(ADR(_awsPublishTopic[iI]),  ADR(_awsPublishTopic[iI + 1]),  SIZEOF(_awsPublishTopic[iI + 1]));
        MEM.MemMove(ADR(_asPublishMessage[iI]), ADR(_asPublishMessage[iI + 1]), SIZEOF(_asPublishMessage[iI + 1]));
    END_FOR

    // Write the new entry into position 0 and safely null-terminate it.
    MEM.MemFill(ADR(_awsPublishTopic[0]),  SIZEOF(_awsPublishTopic[0]),  16#00);
    MEM.MemMove(ADR(wsTopic),              ADR(_awsPublishTopic[0]),     SIZEOF(wsTopic));
    TERMINATE_STRING(psIn := ADR(_awsPublishTopic[0]), udiLength := SIZEOF(wsTopic) - 1);

    MEM.MemFill(ADR(_asPublishMessage[0]), SIZEOF(_asPublishMessage[0]), 16#00);
    MEM.MemMove(ADR(sMessage),             ADR(_asPublishMessage[0]),    SIZEOF(sMessage));
    TERMINATE_STRING(psIn := ADR(_asPublishMessage[0]), udiLength := SIZEOF(sMessage) - 1);

    pushFifoPublish := TRUE;
ELSE
    pushFifoPublish := FALSE;
END_IF

// Watermark for diagnostics.
IF _iFifoPos > _iFifoPosMax THEN
    _iFifoPosMax := _iFifoPos;
END_IF
END_METHOD

END_FUNCTION_BLOCK

// xlh_base/app/IoT/DEVICES/_000_FB_VISU_BASE
// =============================================================================
// _000_FB_VISU_BASE
// -----------------------------------------------------------------------------
// Visualization base FB. Provides a label string (sLabel) and a collection
// of local "dummy" variables that derived FBs use to make values accessible
// for online watch / trace without having to reference them explicitly in
// method bodies.
//
// IMPLEMENTS IVisu — marker interface for all POUs with a visualization.
// =============================================================================
FUNCTION_BLOCK _000_FB_VISU_BASE IMPLEMENTS IVisu
VAR_INPUT
    sLabel : STRING(255) := '';     // Label for the visualization
END_VAR
VAR
    // Helper variables for online watch / trace recordings.
    _bDummy  : BOOL;
    _iDummy  : INT;
    _rDummy  : REAL;
    _fDummy  : LREAL;
    _sDummy  : STRING(GC.STRING_SIZE_MESSAGE_RX);
    _wsDummy : WSTRING(GC.STRING_SIZE_TOPIC);
END_VAR

// No cyclic code — the body stays empty; derived FBs implement their own
// logic.

END_FUNCTION_BLOCK

// xlh_base/app/LOGIC
PROGRAM LOGIC
VAR
	
	fbLampSwitch1: FB_IMPULSE_SWITCH;
	fbLampSwitch2: FB_IMPULSE_SWITCH;
	fbPlug1: FB_IMPULSE_SWITCH;
	fbPlug2: FB_IMPULSE_SWITCH;
	fbShelly1: FB_IMPULSE_SWITCH;
END_VAR

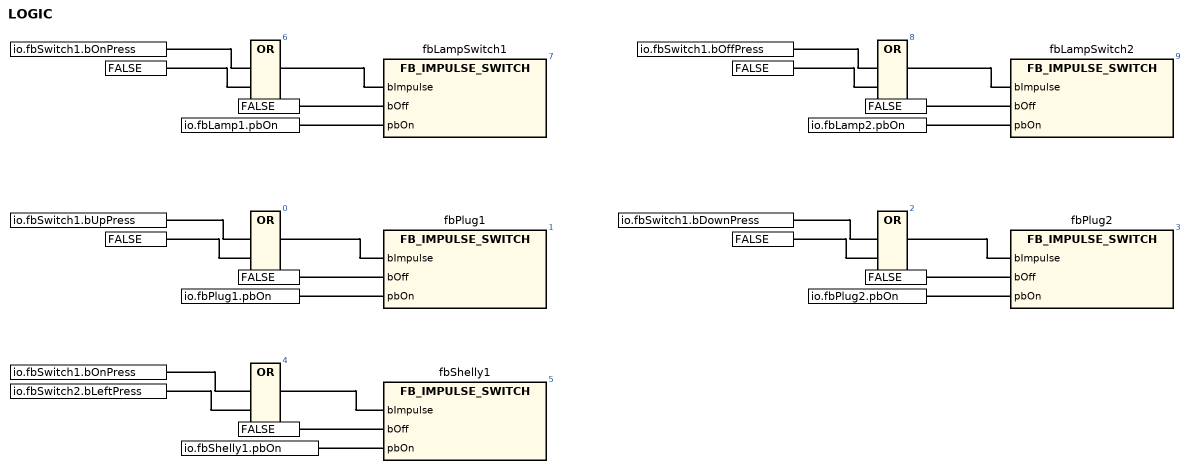
fbPlug1(bImpulse := io.fbSwitch1.bUpPress OR FALSE, bOff := FALSE, pbOn := io.fbPlug1.pbOn); // FB_IMPULSE_SWITCH
fbPlug2(bImpulse := io.fbSwitch1.bDownPress OR FALSE, bOff := FALSE, pbOn := io.fbPlug2.pbOn); // FB_IMPULSE_SWITCH
fbShelly1(
    bImpulse := io.fbSwitch1.bOnPress OR io.fbSwitch2.bLeftPress,
    bOff := FALSE,
    pbOn := io.fbShelly1.pbOn); // FB_IMPULSE_SWITCH
fbLampSwitch1(bImpulse := io.fbSwitch1.bOnPress OR FALSE, bOff := FALSE, pbOn := io.fbLamp1.pbOn); // FB_IMPULSE_SWITCH
fbLampSwitch2(bImpulse := io.fbSwitch1.bOffPress OR FALSE, bOff := FALSE, pbOn := io.fbLamp2.pbOn); // FB_IMPULSE_SWITCH

END_PROGRAM

// xlh_base/app/IoT/FUNCTIONS/FB_IMPULSE_SWITCH
// =============================================================================
// FB_IMPULSE_SWITCH
// -----------------------------------------------------------------------------
// Impulse switch (latching relay) with push-button and impulse inputs as
// well as additional ON/OFF inputs, a maximum on-time and an impulse
// memory.
//
// Behavior:
//   - bImpulse:  A rising edge toggles the state. Sets bImpulseMemory so
//                that subsequent button operations with a falling edge do
//                not switch off.
//   - bButton:   A rising edge switches on. A falling edge switches off,
//                UNLESS bImpulseMemory is set.
//   - bOn:       Forces ON.
//   - bOff:      Forces OFF.
//   - bEnable:   FALSE -> forces OFF and blocks all other actions.
//   - tTimeOnMax:           Maximum on-time; afterwards automatic OFF.
//   - tTimeImpulseMemory:   Lifetime of the impulse memory; afterwards
//                           bImpulseMemory is reset (even in the ON state).
//
// Writes directly to the external variable pointed to by pbOn — this way
// the impulse switch can let several independent inputs act on one shared
// setpoint variable.
// =============================================================================
FUNCTION_BLOCK FB_IMPULSE_SWITCH
VAR_INPUT
    bImpulse           : BOOL;                 // Toggle on rising edge
    bButton            : BOOL;                 // Button pattern (ON while pressed, OFF on release)
    bEnable            : BOOL := TRUE;         // FALSE -> forces OFF
    bOn                : BOOL;                 // Forces ON (static)
    bOff               : BOOL;                 // Forces OFF (static)
    tTimeOnMax         : TIME := T#120M;       // Maximum on-time
    tTimeImpulseMemory : TIME := T#60M;        // Lifetime of the impulse memory
    pbOn               : POINTER TO BOOL;      // Pointer to the setpoint flag (managed externally)
END_VAR
VAR
    bImpulseMemory      : BOOL;     // Protects the ON state from the falling button edge
    fbRtButton          : R_TRIG;
    fbFtButton          : F_TRIG;
    fbTonOnMax          : TON;      // Maximum on-time watchdog
    fbTonImpulseMemory  : TON;      // Lifetime of the impulse memory
END_VAR

// Do nothing without an external setpoint variable.
IF pbOn = 0 THEN
    RETURN;
END_IF

// Evaluate the button pattern.
fbRtButton(CLK := bButton);
IF fbRtButton.Q THEN
    pbOn^ := TRUE;
END_IF

fbFtButton(CLK := bButton);
IF fbFtButton.Q AND NOT bImpulseMemory THEN
    pbOn^ := FALSE;
END_IF

// Toggle impulse.
IF bImpulse THEN
    bImpulseMemory := TRUE;
    pbOn^ := NOT pbOn^;
END_IF

// Static commands.
IF bOn THEN
    pbOn^ := TRUE;
END_IF

IF bOff THEN
    pbOn^ := FALSE;
END_IF

// Maximum on-time.
fbTonOnMax(IN := pbOn^ AND bEnable, PT := tTimeOnMax);
IF fbTonOnMax.Q THEN
    pbOn^ := FALSE;
END_IF

// Reset the impulse memory when the state is already OFF or its lifetime
// has been exceeded.
fbTonImpulseMemory(IN := bImpulseMemory, PT := tTimeImpulseMemory);
IF NOT pbOn^ OR fbTonImpulseMemory.Q THEN
    bImpulseMemory := FALSE;
END_IF

// Device disabled -> forced OFF.
IF NOT bEnable THEN
    pbOn^ := FALSE;
END_IF

END_FUNCTION_BLOCK

// xlh_base/app/IoT/DEVICES/IVisu
// =============================================================================
// IVisu
// -----------------------------------------------------------------------------
// Marker interface for all POUs with a visualization (implemented by
// _000_FB_VISU_BASE).
// =============================================================================
INTERFACE IVisu

END_INTERFACE

// xlh_base/app/IoT/DEVICES/IDevice
// =============================================================================
// IDevice
// -----------------------------------------------------------------------------
// Marker interface for all MQTT device FBs (implemented by _100_FB_DEVICE).
// =============================================================================
INTERFACE IDevice

END_INTERFACE

// xlh_base/app/IoT/MQTT_Client/TERMINATE_STRING
// =============================================================================
// TERMINATE_STRING
// -----------------------------------------------------------------------------
// Writes a null terminator (0x00) at the position defined by udiLength
// within a string buffer.
//
// Usage: the MQTT subscriber returns payloads without a null terminator —
// this function ensures a safe C-style termination so that string
// operations (Stu.StrFind, LEN, ...) work correctly.
//
// Note: the caller is responsible for udiLength being within the buffer
// bounds.
// =============================================================================
FUNCTION TERMINATE_STRING : BOOL
VAR_INPUT
    psIn      : POINTER TO BYTE; // Pointer to the (W)STRING buffer
    udiLength : UDINT;           // Position of the null terminator to insert (byte offset)
END_VAR

psIn[udiLength] := 0;
TERMINATE_STRING := TRUE;

END_FUNCTION

// xlh_base/app/IoT/DEVICES/IDeviceZigbee2Mqtt
// =============================================================================
// IDeviceZigbee2Mqtt
// -----------------------------------------------------------------------------
// Marker interface for Zigbee2MQTT devices (implemented by
// _300_FB_DEVICE_Z2M_BASE).
// =============================================================================
INTERFACE IDeviceZigbee2Mqtt

END_INTERFACE

// xlh_base/app/IoT/MQTT_Client/GET_INT_FROM_VALUE
// =============================================================================
// GET_INT_FROM_VALUE
// -----------------------------------------------------------------------------
// Converts a string value extracted by GET_VALUE_FROM_MSG to INT.
// For an empty input string, the previous value (iValue) is returned
// unchanged.
// =============================================================================
FUNCTION GET_INT_FROM_VALUE : INT
VAR_INPUT
    iValue : INT;           // Previous value (fallback)
    sValue : STRING(255);   // New value as string (e.g. from GET_VALUE_FROM_MSG)
END_VAR

IF sValue <> '' THEN
    iValue := STRING_TO_INT(sValue);
END_IF

GET_INT_FROM_VALUE := iValue;

END_FUNCTION

// xlh_base/app/IoT/MQTT_Client/GET_VALUE_FROM_MSG
// =============================================================================
// GET_VALUE_FROM_MSG
// -----------------------------------------------------------------------------
// Extracts the value of a JSON property from a received MQTT message.
//
// Searches for the pattern `"sKey":` and returns the value up to the next
// separator ',' or '}'. Strings (surrounded by '"') are returned without
// the enclosing quotes.
//
// Limitations:
//   - Simple string parsing, not a full JSON implementation.
//   - Nested objects can be read via the suffix trick in the key,
//     e.g. sKey := 'temperature":{"tC' for {"temperature":{"tC":21.0}}.
//   - Value not found -> returns ''.
// =============================================================================
FUNCTION GET_VALUE_FROM_MSG : STRING(255)
VAR_INPUT
    sKey               : STRING(255);                              // JSON key (without quotes)
    pSubscribedMessage : POINTER TO STRING(GC.STRING_SIZE_MESSAGE_RX); // Received MQTT message
END_VAR
VAR
    iPosKey   : INT;             // Position of the key within the message
    iPosColon : INT;             // Position of the ':' after the key
    iPosEnd   : INT;             // Position of the value end (',' or '}')
    sMessage  : STRING(255);     // Slice of the message starting at the found key
    sValue    : STRING(255);     // Result
END_VAR

// Build the search pattern: "sKey":

sKey := CONCAT(CONCAT('"', sKey), '":');

// Find the position of the key within the whole message and copy the slice.
iPosKey := MAX(0, Stu.StrFindA(pst1:=pSubscribedMessage, pst2:=ADR(sKey), uiSearchStart:=0));
Stu.StrCpyA(pBuffer    := ADR(sMessage),
            iBufferSize:= SIZEOF(sMessage) - 50,
            pStr       := pSubscribedMessage + INT_TO_DWORD(iPosKey));

// Find the position of the ':' after the key (value start) and of the next
// separator (',' or '}').
iPosColon := MAX(0, Stu.StrFindA(pst1:=ADR(sMessage),
                                 pst2:=ADR(':'),
                                 uiSearchStart:=INT_TO_UINT(MAX(0, LEN(sKey) - 1))));
iPosEnd   := MAX(0, Stu.StrFindA(pst1:=ADR(sMessage),
                                 pst2:=ADR(','),
                                 uiSearchStart:=INT_TO_UINT(MAX(0, LEN(sKey)))));
IF iPosEnd = 0 THEN
    iPosEnd := MAX(0, Stu.StrFindA(pst1:=ADR(sMessage),
                                   pst2:=ADR('}'),
                                   uiSearchStart:=INT_TO_UINT(MAX(0, LEN(sKey)))));
END_IF

// Extract the value if the key and the separator were found.
// (MID/LEFT only work for strings with length < 255.)
IF (iPosColon <> 0) AND (iPosEnd <> 0) THEN
    sValue := MID(sMessage, iPosEnd - iPosColon - 1, iPosColon + 1);
    // Remove the quotes if the value is a string.
    IF LEFT(sMessage, 1) = '"' THEN
        sValue := MID(sValue, LEN(sValue) - 2, 2);
    END_IF
ELSE
    sValue := '';
END_IF

GET_VALUE_FROM_MSG := sValue;

END_FUNCTION

// xlh_base/app/IoT/MQTT_Client/GET_STRING_FROM_VALUE
// =============================================================================
// GET_STRING_FROM_VALUE
// -----------------------------------------------------------------------------
// Returns a string value extracted by GET_VALUE_FROM_MSG without the
// enclosing quotes.
// For an empty input string, the previous value (sValuePrev) is returned
// unchanged.
// =============================================================================
FUNCTION GET_STRING_FROM_VALUE : STRING(255)
VAR_INPUT
    sValuePrev : STRING(255);   // Previous value (fallback)
    sValue     : STRING(255);   // New value as string (e.g. from GET_VALUE_FROM_MSG)
END_VAR
VAR
    sResult : STRING(255);
END_VAR

// Keep the previous value by default.

sResult := sValuePrev;

// Take over the new value if present.
IF sValue <> '' THEN
    sResult := sValue;
END_IF

// Remove the quotes at the beginning and end (e.g. '"abc"' -> 'abc').
IF LEN(sValue) > 2 THEN
    sResult := LEFT(sResult, LEN(sValue) - 1);
    sResult := RIGHT(sResult, LEN(sValue) - 2);
END_IF

GET_STRING_FROM_VALUE := sResult;

END_FUNCTION

// xlh_base/app/IoT/DEVICES/_345_FB_DEVICE_Z2M_BATTERY_HUE_WALL_SWITCH
// =============================================================================
// _345_FB_DEVICE_Z2M_BATTERY_HUE_WALL_SWITCH
// -----------------------------------------------------------------------------
// Philips Hue Wall Switch Module — 2-channel wireless switch (left / right)
// with press / hold / release actions per button.
// Device link: https://www.zigbee2mqtt.io/devices/929003017102.html
//
// Behavior of the boolean outputs:
//   - Pulses: set for EXACTLY ONE PLC cycle when an action is received,
//     reset again in the following cycle.
// =============================================================================
FUNCTION_BLOCK _345_FB_DEVICE_Z2M_BATTERY_HUE_WALL_SWITCH EXTENDS _340_FB_DEVICE_Z2M_BATTERY
VAR_OUTPUT
    sAction            : STRING(255);   // Last reported action (diagnostics)

    // Left button
    bLeftPress         : BOOL;
    bLeftPressRelease  : BOOL;
    bLeftHold          : BOOL;
    bLeftHoldRelease   : BOOL;

    // Right button
    bRightPress        : BOOL;
    bRightPressRelease : BOOL;
    bRightHold         : BOOL;
    bRightHoldRelease  : BOOL;
END_VAR
VAR
    _bNewAction : BOOL;
END_VAR

SUPER^();

IF _bNewAction THEN
    _bNewAction := FALSE;

    bLeftPress         := sAction = 'left_press';
    bLeftPressRelease  := sAction = 'left_press_release';
    bLeftHold          := sAction = 'left_hold';
    bLeftHoldRelease   := sAction = 'left_hold_release';

    bRightPress        := sAction = 'right_press';
    bRightPressRelease := sAction = 'right_press_release';
    bRightHold         := sAction = 'right_hold';
    bRightHoldRelease  := sAction = 'right_hold_release';
ELSE
    bLeftPress         := FALSE;
    bLeftPressRelease  := FALSE;
    bLeftHold          := FALSE;
    bLeftHoldRelease   := FALSE;

    bRightPress        := FALSE;
    bRightPressRelease := FALSE;
    bRightHold         := FALSE;
    bRightHoldRelease  := FALSE;
END_IF

// =============================================================================
// METHOD newMessage
// -----------------------------------------------------------------------------
// Reads the action from the event topic and triggers the pulse logic in
// the next cycle.
// =============================================================================
METHOD newMessage : BOOL
SUPER^.newMessage();
IF _fbMqttSubscriber.wsLastTopic = _wsMqttTopicEvent THEN
    sAction := GET_STRING_FROM_VALUE(sAction, GET_VALUE_FROM_MSG('action', ADR(_sSubscribedMessage)));
    THIS^._bNewAction := TRUE;
END_IF
END_METHOD

END_FUNCTION_BLOCK

// xlh_base/app/IoT/DEVICES/_341_FB_DEVICE_Z2M_BATTERY_SONOFF_TEMP_HUM
// =============================================================================
// _341_FB_DEVICE_Z2M_BATTERY_SONOFF_TEMP_HUM
// -----------------------------------------------------------------------------
// Sonoff SNZB-02D — temperature and humidity sensor with display.
// Device link: https://www.zigbee2mqtt.io/devices/SNZB-02D.html
//
// Offers an offset correction (fParTemperatureOffset / fParHumidityOffset)
// for the calibration-free adjustment to reference devices.
//
// Example message (event):
//   {"battery":100,"humidity":52.4,"linkquality":174,
//    "temperature":20.5,"temperature_units":"celsius", ...}
// =============================================================================
FUNCTION_BLOCK _341_FB_DEVICE_Z2M_BATTERY_SONOFF_TEMP_HUM EXTENDS _340_FB_DEVICE_Z2M_BATTERY
VAR_INPUT
    fParTemperatureOffset : LREAL := 0.0;   // Offset on the temperature reading (°C)
    fParHumidityOffset    : LREAL := 0.0;   // Offset on the humidity reading (%)
END_VAR
VAR_OUTPUT
    fTemperature : LREAL := -1.0;           // Temperature (°C, incl. offset)
    fHumidity    : LREAL := -1.0;           // Relative humidity (%, incl. offset)
END_VAR

SUPER^();

// =============================================================================
// METHOD newMessage
// -----------------------------------------------------------------------------
// Reads temperature and humidity from the event topic and adds the
// configured offsets.
// =============================================================================
METHOD newMessage : BOOL
SUPER^.newMessage();
IF _fbMqttSubscriber.wsLastTopic = _wsMqttTopicEvent THEN
    fTemperature := GET_LREAL_FROM_VALUE(fTemperature, GET_VALUE_FROM_MSG('temperature', ADR(_sSubscribedMessage))) + fParTemperatureOffset;
    fHumidity    := GET_LREAL_FROM_VALUE(fHumidity,    GET_VALUE_FROM_MSG('humidity',    ADR(_sSubscribedMessage))) + fParHumidityOffset;
END_IF
END_METHOD

END_FUNCTION_BLOCK

// xlh_base/app/IoT/MQTT_Client/GET_LREAL_FROM_VALUE
// =============================================================================
// GET_LREAL_FROM_VALUE
// -----------------------------------------------------------------------------
// Converts a string value extracted by GET_VALUE_FROM_MSG to LREAL.
// For an empty input string, the previous value (fValue) is returned
// unchanged.
// =============================================================================
FUNCTION GET_LREAL_FROM_VALUE : LREAL
VAR_INPUT
    fValue : LREAL;         // Previous value (fallback)
    sValue : STRING(255);   // New value as string (e.g. from GET_VALUE_FROM_MSG)
END_VAR

IF sValue <> '' THEN
    fValue := STRING_TO_LREAL(sValue);
END_IF

GET_LREAL_FROM_VALUE := fValue;

END_FUNCTION

// xlh_base/app/IoT/DEVICES/_344_FB_DEVICE_Z2M_BATTERY_HUE_MOTION
// =============================================================================
// _344_FB_DEVICE_Z2M_BATTERY_HUE_MOTION
// -----------------------------------------------------------------------------
// Philips Hue Outdoor Motion Sensor — motion, illuminance, temperature.
// Device link: https://www.zigbee2mqtt.io/devices/9290030675.html
//
// Logic:
//   - bOccupancy        : Raw motion report from the sensor.
//   - bOccupancyDelay   : Motion with a configurable off-delay (TOF).
//   - bOccupancyDelayTod: bOccupancyDelay additionally gated by the time
//                         of day (between todEnableStart and todEnableEnd,
//                         across midnight).
//
// Example message (event):
//   {"battery":16.5,"illuminance":15,"linkquality":188,
//    "occupancy":false,"occupancy_timeout":3,"temperature":21.06, ...}
// =============================================================================
FUNCTION_BLOCK _344_FB_DEVICE_Z2M_BATTERY_HUE_MOTION EXTENDS _340_FB_DEVICE_Z2M_BATTERY
VAR_INPUT
    fParTemperatureOffset : LREAL       := 0.0;        // Offset on the temperature (°C)
    fParIlluminanceOffset : LREAL       := 0.0;        // Offset on the illuminance (lux)
    tDelay                : TIME        := T#5S;      // Off-delay for bOccupancyDelay
    todEnableStart        : TIME_OF_DAY := TOD#18:00;  // Start of the active window (may span midnight)
    todEnableEnd          : TIME_OF_DAY := TOD#8:00;   // End of the active window
END_VAR
VAR_OUTPUT
    bOccupancy        : BOOL  := FALSE; // Current motion report
    bOccupancyDelay   : BOOL  := FALSE; // bOccupancy with off-delay
    bOccupancyDelayTod: BOOL  := FALSE; // bOccupancyDelay AND active window
    fTemperature      : LREAL := -1.0;  // Temperature (°C, incl. offset)
    fIlluminance      : LREAL := -1.0;  // Illuminance (lux, incl. offset)
END_VAR
VAR
    fbTofDelay  : TOF;          // Off-delay for bOccupancyDelay
    bEnableTod  : BOOL;         // TRUE during the active window
END_VAR

SUPER^();

// Off-delay on the motion report.
fbTofDelay(IN := bOccupancy, PT := tDelay, Q => bOccupancyDelay);

// Active window across midnight: [todEnableStart .. 23:59:59.999]
//                             OR [00:00:00.000 .. todEnableEnd]
bEnableTod :=     (LOCAL_TIME_AND_TIME_ZONE.todTime >= todEnableStart)
              AND (LOCAL_TIME_AND_TIME_ZONE.todTime <= TOD#23:59:59.999)
           OR     (LOCAL_TIME_AND_TIME_ZONE.todTime <= todEnableEnd)
              AND (LOCAL_TIME_AND_TIME_ZONE.todTime >= TOD#00:00:00.000);

//bOccupancyDelayTod := bOccupancyDelay AND bEnableTod;
bOccupancyDelayTod := bOccupancyDelay;

// =============================================================================
// METHOD newMessage
// -----------------------------------------------------------------------------
// Reads occupancy, temperature and illuminance from the event topic.
// =============================================================================
METHOD newMessage : BOOL
SUPER^.newMessage();
IF _fbMqttSubscriber.wsLastTopic = _wsMqttTopicEvent THEN
    bOccupancy   := GET_BOOL_FROM_VALUE (bOccupancy,   GET_VALUE_FROM_MSG('occupancy',   ADR(_sSubscribedMessage)));
    fTemperature := GET_LREAL_FROM_VALUE(fTemperature, GET_VALUE_FROM_MSG('temperature', ADR(_sSubscribedMessage))) + fParTemperatureOffset;
    fIlluminance := GET_LREAL_FROM_VALUE(fIlluminance, GET_VALUE_FROM_MSG('illuminance', ADR(_sSubscribedMessage))) + fParIlluminanceOffset;
END_IF
END_METHOD

END_FUNCTION_BLOCK

// xlh_base/app/IoT/MQTT_Client/GET_BOOL_FROM_VALUE
// =============================================================================
// GET_BOOL_FROM_VALUE
// -----------------------------------------------------------------------------
// Converts a string value extracted by GET_VALUE_FROM_MSG to BOOL.
// Expects the JSON format in lower case ('true'/'false').
// For an empty input string, the previous value (bValue) is returned
// unchanged.
// =============================================================================
FUNCTION GET_BOOL_FROM_VALUE : BOOL
VAR_INPUT
    bValue : BOOL;          // Previous value (fallback)
    sValue : STRING(255);   // New value as string (e.g. from GET_VALUE_FROM_MSG)
END_VAR

IF sValue <> '' THEN
    bValue := (sValue = 'true');
END_IF

GET_BOOL_FROM_VALUE := bValue;

END_FUNCTION

// xlh_base/app/IoT/DEVICES/_312_FB_DEVICE_Z2M_POWER_LAMP
// =============================================================================
// _312_FB_DEVICE_Z2M_POWER_LAMP
// -----------------------------------------------------------------------------
// Zigbee2MQTT lamp with brightness and color temperature (color_temp).
// Example: IKEA TRADFRI bulb.
//
// Request/status concept:
//   - Values received from the Z2M event are mirrored into iBrightness,
//     iColorTemp and iColorTempStartup AND recorded as the written value.
//   - On an external change (e.g. via the visualization), the publisher
//     pushes the values to the device via <z2m>/<base>/set.
//
// Example message (event):
//   {"brightness":6,"color_mode":"color_temp","color_temp":454,
//    "color_temp_startup":250,"linkquality":109,
//    "power_on_behavior":"off","state":"ON", ...}
// =============================================================================
FUNCTION_BLOCK _312_FB_DEVICE_Z2M_POWER_LAMP EXTENDS _310_FB_DEVICE_Z2M_POWER_SWITCH
VAR_OUTPUT
    sColorMode         : STRING(255) := 'NONE';   // Active color mode (e.g. 'color_temp')
    iBrightness        : INT := -1;               // Brightness (0..254)
    iColorTemp         : INT := -1;               // Color temperature in mireds
    iColorTempStartup  : INT := -1;               // Startup color temperature after power-up
END_VAR
VAR
    _iBrightnessWrite        : INT := -1;     // Last published setpoint
    _iColorTempWrite         : INT := -1;
    _iColorTempStartupWrite  : INT := -1;
END_VAR

SUPER^();

// =============================================================================
// METHOD newMessage
// -----------------------------------------------------------------------------
// Mirrors the values reported by the device into the outputs AND into the
// written-value variables so the publisher does not trigger a superfluous
// set command.
// =============================================================================
METHOD newMessage : BOOL
SUPER^.newMessage();
IF _fbMqttSubscriber.wsLastTopic = _wsMqttTopicEvent THEN
    sColorMode        := GET_STRING_FROM_VALUE(sColorMode,        GET_VALUE_FROM_MSG('color_mode',         ADR(_sSubscribedMessage)));
    iBrightness       := GET_INT_FROM_VALUE   (iBrightness,       GET_VALUE_FROM_MSG('brightness',         ADR(_sSubscribedMessage)));
    iColorTemp        := GET_INT_FROM_VALUE   (iColorTemp,        GET_VALUE_FROM_MSG('color_temp',         ADR(_sSubscribedMessage)));
    iColorTempStartup := GET_INT_FROM_VALUE   (iColorTempStartup, GET_VALUE_FROM_MSG('color_temp_startup', ADR(_sSubscribedMessage)));

    // Take over the actual values as last written so the publisher does
    // not react to them as a "change" again.
    _iBrightnessWrite       := iBrightness;
    _iColorTempWrite        := iColorTemp;
    _iColorTempStartupWrite := iColorTempStartup;
END_IF
END_METHOD

// =============================================================================
// METHOD publisher
// -----------------------------------------------------------------------------
// Writes changed brightness / color-temperature setpoints as individual
// JSON properties to <z2m>/<base>/set.
// =============================================================================
METHOD publisher : BOOL
VAR
    sPublishMessage     : STRING(GC.STRING_SIZE_MESSAGE_TX);
    sPublishMessageTemp : STRING(255);
END_VAR

// Update the brightness.
IF THIS^._iBrightnessWrite <> THIS^.iBrightness THEN
    sPublishMessage     := '{"brightness": ';
    sPublishMessageTemp := TO_STRING(THIS^.iBrightness);
    Stu.StrConcatA(pstFrom:=ADR(sPublishMessageTemp), pstTo:=ADR(sPublishMessage), iBufferSize:=GC.STRING_SIZE_MESSAGE_TX);
    Stu.StrConcatA(pstFrom:=ADR('}'),                 pstTo:=ADR(sPublishMessage), iBufferSize:=GC.STRING_SIZE_MESSAGE_TX);
    THIS^.pushFifoPublish(THIS^._wsMqttTopicSet, sPublishMessage);
    THIS^._iBrightnessWrite := THIS^.iBrightness;
END_IF

// Update the color temperature.
IF THIS^._iColorTempWrite <> THIS^.iColorTemp THEN
    sPublishMessage     := '{"color_temp": ';
    sPublishMessageTemp := TO_STRING(THIS^.iColorTemp);
    Stu.StrConcatA(pstFrom:=ADR(sPublishMessageTemp), pstTo:=ADR(sPublishMessage), iBufferSize:=GC.STRING_SIZE_MESSAGE_TX);
    Stu.StrConcatA(pstFrom:=ADR('}'),                 pstTo:=ADR(sPublishMessage), iBufferSize:=GC.STRING_SIZE_MESSAGE_TX);
    THIS^.pushFifoPublish(THIS^._wsMqttTopicSet, sPublishMessage);
    THIS^._iColorTempWrite := THIS^.iColorTemp;
END_IF

// Update the startup color temperature.
IF THIS^._iColorTempStartupWrite <> THIS^.iColorTempStartup THEN
    sPublishMessage     := '{"color_temp_startup": ';
    sPublishMessageTemp := TO_STRING(THIS^.iColorTempStartup);
    Stu.StrConcatA(pstFrom:=ADR(sPublishMessageTemp), pstTo:=ADR(sPublishMessage), iBufferSize:=GC.STRING_SIZE_MESSAGE_TX);
    Stu.StrConcatA(pstFrom:=ADR('}'),                 pstTo:=ADR(sPublishMessage), iBufferSize:=GC.STRING_SIZE_MESSAGE_TX);
    THIS^.pushFifoPublish(THIS^._wsMqttTopicSet, sPublishMessage);
    THIS^._iColorTempStartupWrite := THIS^.iColorTempStartup;
END_IF

SUPER^.publisher();
END_METHOD

END_FUNCTION_BLOCK

// xlh_base/app/IoT/DEVICES/_310_FB_DEVICE_Z2M_POWER_SWITCH
// =============================================================================
// _310_FB_DEVICE_Z2M_POWER_SWITCH
// -----------------------------------------------------------------------------
// Generic Zigbee2MQTT switch actuator (e.g. plug, relay).
//
// Functionality:
//   - Writes {"state":"ON"|"OFF"} to <z2m>/<base>/set when the request bOn
//     changes or differs from the reported actual state bOnState for longer
//     than _tACTION_TIME_NOT_EQUAL.
//   - Periodic status query every _fREFRESH_TIME seconds via {"state":""}
//     on <z2m>/<base>/get.
//   - Provides a pointer pbOn to the request so that external logic (see
//     LOGIC.FB_IMPULSE_SWITCH) can set the setpoint directly.
//
// Example message (event):
//   {"current":0.03,"energy":0,"linkquality":160,"power":0,
//    "power_on_behavior":"off","state":"OFF",
//    "update":{"installed_version":...,"latest_version":...,"state":"idle"},
//    "voltage":0.1}
// =============================================================================
FUNCTION_BLOCK _310_FB_DEVICE_Z2M_POWER_SWITCH EXTENDS _300_FB_DEVICE_Z2M_BASE
VAR_INPUT
    bOn : BOOL;                                     // Request
END_VAR
VAR_OUTPUT
    pbOn               : POINTER TO BOOL;           // Pointer to bOn (for external logic)
    sPowerOnBehavior   : STRING(255) := 'zigbee2mqtt'; // Behavior after a power failure (device parameter)
    bOnState           : BOOL;                      // Actual state (reported by the device)
END_VAR
VAR
    _fbRtRelais             : R_TRIG;
    _fbFtRelais             : F_TRIG;
    _fbTonDiffRelaisState   : TON;          // Watchdog: request <> state for longer than _tACTION_TIME_NOT_EQUAL
    _fTimer                 : LREAL := 0.0; // Second counter for the periodic status query
END_VAR
VAR CONSTANT
    _tACTION_TIME_NOT_EQUAL : TIME  := T#1000MS;
    _fREFRESH_TIME          : LREAL := 300.0;
END_VAR

SUPER^();

// Periodic status query.
_fTimer := LIMIT(0.0, _fTimer + TASK_INFO.fCycleTime, 99999.0);
IF _fTimer >= _fREFRESH_TIME THEN
    _fTimer := 0.0;
    statusUpdate();
END_IF

// =============================================================================
// METHOD statusUpdate
// -----------------------------------------------------------------------------
// Forces a status response by sending {"state":""} to <z2m>/<base>/get.
// =============================================================================
METHOD statusUpdate : BOOL
VAR
    sPublishMessage : STRING(GC.STRING_SIZE_MESSAGE_TX);
END_VAR
SUPER^.statusUpdate();
sPublishMessage := '{"state":""}';
THIS^.pushFifoPublish(THIS^._wsMqttTopicGet, sPublishMessage);
END_METHOD

// =============================================================================
// METHOD startup
// -----------------------------------------------------------------------------
// Sets the external pointer pbOn and initializes _fTimer so that an
// immediate status query is made in the first cycle.
// =============================================================================
METHOD startup : BOOL
SUPER^.startup();
THIS^.pbOn    := ADR(THIS^.bOn);
THIS^._fTimer := THIS^._fREFRESH_TIME - 1.0;     // Trigger the first query promptly.
END_METHOD

// =============================================================================
// METHOD newMessage
// -----------------------------------------------------------------------------
// Reads power_on_behavior and state from the Z2M event topic.
// =============================================================================
METHOD newMessage : BOOL
SUPER^.newMessage();
IF _fbMqttSubscriber.wsLastTopic = _wsMqttTopicEvent THEN
    sPowerOnBehavior := GET_STRING_FROM_VALUE     (sPowerOnBehavior, GET_VALUE_FROM_MSG('power_on_behavior', ADR(_sSubscribedMessage)));
    bOnState         := GET_BOOL_FROM_VALUE_ON_OFF(bOnState,         GET_VALUE_FROM_MSG('state',             ADR(_sSubscribedMessage)));
END_IF
END_METHOD

// =============================================================================
// METHOD publisher
// -----------------------------------------------------------------------------
// Publishes the requested state to <z2m>/<base>/set when bOn changes or
// differs from the actual state for too long.
// =============================================================================
METHOD publisher : BOOL
VAR
    bPublishState   : BOOL;
    sPublishMessage : STRING(GC.STRING_SIZE_MESSAGE_TX);
END_VAR
THIS^._fbTonDiffRelaisState(IN := ((THIS^.bOn <> THIS^.bOnState) AND NOT _fbTonDiffRelaisState.Q),
                            PT := THIS^._tACTION_TIME_NOT_EQUAL);
THIS^._fbRtRelais(CLK := THIS^.bOn);
THIS^._fbFtRelais(CLK := THIS^.bOn);
bPublishState := _fbTonDiffRelaisState.Q OR _fbRtRelais.Q OR _fbFtRelais.Q;

IF bPublishState THEN
    IF THIS^.bOn THEN
        sPublishMessage := '{"state": "ON"}';
    ELSE
        sPublishMessage := '{"state": "OFF"}';
    END_IF
    THIS^.pushFifoPublish(THIS^._wsMqttTopicSet, sPublishMessage);
END_IF

SUPER^.publisher();
END_METHOD

END_FUNCTION_BLOCK

// xlh_base/app/IoT/MQTT_Client/GET_BOOL_FROM_VALUE_ON_OFF
// =============================================================================
// GET_BOOL_FROM_VALUE_ON_OFF
// -----------------------------------------------------------------------------
// Converts a string value extracted by GET_VALUE_FROM_MSG to BOOL.
// Expects the Zigbee2MQTT convention in upper case ('"ON"'/'"OFF"').
// For an empty input string, the previous value (bValue) is returned
// unchanged.
// =============================================================================
FUNCTION GET_BOOL_FROM_VALUE_ON_OFF : BOOL
VAR_INPUT
    bValue : BOOL;          // Previous value (fallback)
    sValue : STRING(255);   // New value as string (e.g. from GET_VALUE_FROM_MSG)
END_VAR

IF sValue <> '' THEN
    bValue := (sValue = '"ON"');
END_IF

GET_BOOL_FROM_VALUE_ON_OFF := bValue;

END_FUNCTION

// xlh_base/app/IoT/DEVICES/_311_FB_DEVICE_Z2M_POWER_SWITCH_IKEA_INSPELING
// =============================================================================
// _311_FB_DEVICE_Z2M_POWER_SWITCH_IKEA_INSPELING
// -----------------------------------------------------------------------------
// IKEA INSPELNING (E2206) smart plug with energy metering.
// Extends _310 with the measurement outputs for power, voltage, current
// and energy.
//
// Device link: https://www.zigbee2mqtt.io/devices/E2206.html
//
// Example message (event):
//   {"current":0.03,"energy":0,"linkquality":160,"power":0,
//    "power_on_behavior":"off","state":"OFF","voltage":0.1, ...}
// =============================================================================
FUNCTION_BLOCK _311_FB_DEVICE_Z2M_POWER_SWITCH_IKEA_INSPELING EXTENDS _310_FB_DEVICE_Z2M_POWER_SWITCH
VAR_OUTPUT
    fPower   : LREAL;       // Active power (W)
    fVoltage : LREAL;       // Mains voltage (V)
    fCurrent : LREAL;       // Current (A)
    fEnergy  : LREAL;       // Cumulative energy (kWh)
END_VAR

SUPER^();

// =============================================================================
// METHOD newMessage
// -----------------------------------------------------------------------------
// Reads the additional measurements from the Z2M event topic.
// =============================================================================
METHOD newMessage : BOOL
SUPER^.newMessage();
IF _fbMqttSubscriber.wsLastTopic = _wsMqttTopicEvent THEN
    fPower   := GET_LREAL_FROM_VALUE(fPower,   GET_VALUE_FROM_MSG('power',   ADR(_sSubscribedMessage)));
    fVoltage := GET_LREAL_FROM_VALUE(fVoltage, GET_VALUE_FROM_MSG('voltage', ADR(_sSubscribedMessage)));
    fCurrent := GET_LREAL_FROM_VALUE(fCurrent, GET_VALUE_FROM_MSG('current', ADR(_sSubscribedMessage)));
    fEnergy  := GET_LREAL_FROM_VALUE(fEnergy,  GET_VALUE_FROM_MSG('energy',  ADR(_sSubscribedMessage)));
END_IF
END_METHOD

END_FUNCTION_BLOCK

// xlh_base/app/IoT/DEVICES/_313_FB_DEVICE_Z2M_SHELLY_1PM
// =============================================================================
// _313_FB_DEVICE_Z2M_SHELLY_1PM
// -----------------------------------------------------------------------------
// Shelly 1PM, connected via Zigbee2MQTT (not via the native Shelly MQTT
// schema). Behaves like _310 (switch actuator with ON/OFF state) and
// additionally provides measurements for power, voltage, current, energy
// and mains frequency.
//
// Device link: https://www.zigbee2mqtt.io/devices/E2206.html
//
// Example message (event):
//   {"ac_frequency":50.03,"current":0.1,"energy":0,
//    "linkquality":120,"power":31,"state":"ON","voltage":238.68, ...}
// =============================================================================
FUNCTION_BLOCK _313_FB_DEVICE_Z2M_SHELLY_1PM EXTENDS _310_FB_DEVICE_Z2M_POWER_SWITCH
VAR_OUTPUT
    fPower     : LREAL;     // Active power (W)
    fVoltage   : LREAL;     // Mains voltage (V)
    fCurrent   : LREAL;     // Current (A)
    fEnergy    : LREAL;     // Cumulative energy (kWh)
    fFrequency : LREAL;     // Mains frequency (Hz)
END_VAR

SUPER^();

// =============================================================================
// METHOD newMessage
// -----------------------------------------------------------------------------
// Reads the additional measurements from the Z2M event topic.
// =============================================================================
METHOD newMessage : BOOL
SUPER^.newMessage();
IF _fbMqttSubscriber.wsLastTopic = _wsMqttTopicEvent THEN
    fPower     := GET_LREAL_FROM_VALUE(fPower,     GET_VALUE_FROM_MSG('power',        ADR(_sSubscribedMessage)));
    fVoltage   := GET_LREAL_FROM_VALUE(fVoltage,   GET_VALUE_FROM_MSG('voltage',      ADR(_sSubscribedMessage)));
    fCurrent   := GET_LREAL_FROM_VALUE(fCurrent,   GET_VALUE_FROM_MSG('current',      ADR(_sSubscribedMessage)));
    fEnergy    := GET_LREAL_FROM_VALUE(fEnergy,    GET_VALUE_FROM_MSG('energy',       ADR(_sSubscribedMessage)));
    fFrequency := GET_LREAL_FROM_VALUE(fFrequency, GET_VALUE_FROM_MSG('ac_frequency', ADR(_sSubscribedMessage)));
END_IF
END_METHOD

END_FUNCTION_BLOCK

// xlh_base/app/IoT/DEVICES/_314_FB_DEVICE_Z2M_SHELLY_EM
// =============================================================================
// _314_FB_DEVICE_Z2M_SHELLY_EM
// -----------------------------------------------------------------------------
// Shelly EM (energy meter) via Zigbee2MQTT. In contrast to _313 it is not
// a switch actuator — therefore derived directly from _300 without the
// ON/OFF logic.
//
// Example message (event):
//   {"ac_frequency":49.97,"current":0,"energy":0.02,
//    "ip_address":"...","linkquality":140,"power":24,
//    "voltage":237.42, ...}
// =============================================================================
FUNCTION_BLOCK _314_FB_DEVICE_Z2M_SHELLY_EM EXTENDS _300_FB_DEVICE_Z2M_BASE
VAR_OUTPUT
    fPower     : LREAL;     // Active power (W)
    fVoltage   : LREAL;     // Mains voltage (V)
    fCurrent   : LREAL;     // Current (A)
    fEnergy    : LREAL;     // Cumulative energy (kWh)
    fFrequency : LREAL;     // Mains frequency (Hz)
END_VAR

SUPER^();

// =============================================================================
// METHOD newMessage
// -----------------------------------------------------------------------------
// Reads the measurements from the Z2M event topic.
// =============================================================================
METHOD newMessage : BOOL
SUPER^.newMessage();
IF _fbMqttSubscriber.wsLastTopic = _wsMqttTopicEvent THEN
    fPower     := GET_LREAL_FROM_VALUE(fPower,     GET_VALUE_FROM_MSG('power',        ADR(_sSubscribedMessage)));
    fVoltage   := GET_LREAL_FROM_VALUE(fVoltage,   GET_VALUE_FROM_MSG('voltage',      ADR(_sSubscribedMessage)));
    fCurrent   := GET_LREAL_FROM_VALUE(fCurrent,   GET_VALUE_FROM_MSG('current',      ADR(_sSubscribedMessage)));
    fEnergy    := GET_LREAL_FROM_VALUE(fEnergy,    GET_VALUE_FROM_MSG('energy',       ADR(_sSubscribedMessage)));
    fFrequency := GET_LREAL_FROM_VALUE(fFrequency, GET_VALUE_FROM_MSG('ac_frequency', ADR(_sSubscribedMessage)));
END_IF
END_METHOD

END_FUNCTION_BLOCK

// xlh_base/app/MAIN
// =============================================================================
// MAIN
// -----------------------------------------------------------------------------
// Entry point of the MainTask. Calls the LOGIC program, in which the device
// interconnections are modeled graphically (FBD/CFC). The io program and the
// diagnostics programs are called directly by the task (see Task
// Configuration).
// =============================================================================
PROGRAM MAIN
VAR
END_VAR

LOGIC();

END_PROGRAM

// xlh_base/app/IoT/MQTT_Client/GET_REAL_FROM_VALUE
// =============================================================================
// GET_REAL_FROM_VALUE
// -----------------------------------------------------------------------------
// Converts a string value extracted by GET_VALUE_FROM_MSG to REAL.
// For an empty input string, the previous value (rValue) is returned
// unchanged — so previously received data is kept when the property is
// not contained in the current message.
// =============================================================================
FUNCTION GET_REAL_FROM_VALUE : REAL
VAR_INPUT
    rValue : REAL;          // Previous value (fallback)
    sValue : STRING(255);   // New value as string (e.g. from GET_VALUE_FROM_MSG)
END_VAR

IF sValue <> '' THEN
    rValue := STRING_TO_REAL(sValue);
END_IF

GET_REAL_FROM_VALUE := rValue;

END_FUNCTION

// xlh_base/app/IoT/DEVICES/_200_FB_DEVICE_SHELLY_BASE
// =============================================================================
// _200_FB_DEVICE_SHELLY_BASE
// -----------------------------------------------------------------------------
// Base FB for Shelly devices (Plus/Pro generation, JSON-RPC over MQTT).
//
// Topic structure (non-standard Shelly, requires assignment in the device
// configuration):
//   <base>/rpc           -> publish: JSON-RPC requests to the device
//   <base>/events/rpc    -> subscribe: events triggered by the device
//   <base>/status/rpc    -> subscribe: responses to Shelly.GetStatus
//
// Functionality:
//   - Periodic status query (every _fREFRESH_TIME seconds) via
//     statusUpdate() / Shelly.GetStatus.
//   - newMessage() extracts generic fields (temperature, RSSI, SSID, MAC).
// =============================================================================
FUNCTION_BLOCK _200_FB_DEVICE_SHELLY_BASE EXTENDS _100_FB_DEVICE IMPLEMENTS IDeviceShelly
VAR_OUTPUT
    fTemperaturePcb : LREAL;        // Internal temperature of the device (°C)
    sSsid           : STRING(255);  // WLAN SSID
    sMacId          : STRING(255);  // BSSID/MAC of the access point
    iRssi           : INT;          // WLAN signal strength (dBm)
END_VAR
VAR
    _wsMqttTopicEvent  : WSTRING(GC.STRING_SIZE_TOPIC); // <base>/events/rpc
    _wsMqttTopicStatus : WSTRING(GC.STRING_SIZE_TOPIC); // <base>/status/rpc
    _fTimer            : LREAL := 0.0;                  // Second counter for the refresh
END_VAR
VAR CONSTANT
    _fREFRESH_TIME : LREAL := 300.0;   // Periodic status query every 300s
END_VAR

SUPER^();

// Periodic status query.
_fTimer := LIMIT(0.0, _fTimer + TASK_INFO.fCycleTime, 99999.0);
IF _fTimer >= _fREFRESH_TIME THEN
    _fTimer := 0.0;
    statusUpdate();
END_IF

// =============================================================================
// METHOD statusUpdate
// -----------------------------------------------------------------------------
// Sends a Shelly.GetStatus RPC query. The response arrives on
// <base>/status/rpc.
// =============================================================================
METHOD statusUpdate : BOOL
VAR
    sPublishMessage : STRING(GC.STRING_SIZE_MESSAGE_TX);
END_VAR
SUPER^.statusUpdate();

// {"id":1, "src":"<base>/status", "method":"Shelly.GetStatus"}
sPublishMessage := '{"id":1, "src":"';
Stu.StrConcatA(pstFrom:=ADR(THIS^.sMqttTopicBase),                          pstTo:=ADR(sPublishMessage), iBufferSize:=GC.STRING_SIZE_MESSAGE_TX);
Stu.StrConcatA(pstFrom:=ADR('/status", "method":"Shelly.GetStatus"}'),      pstTo:=ADR(sPublishMessage), iBufferSize:=GC.STRING_SIZE_MESSAGE_TX);

THIS^.pushFifoPublish(THIS^._wsPublishTopic, sPublishMessage);
END_METHOD

// =============================================================================
// METHOD startup
// -----------------------------------------------------------------------------
// Initializes the Shelly-specific topics (publish target /rpc, event topic
// /events/rpc, status topic /status/rpc).
// =============================================================================
METHOD startup : BOOL
SUPER^.startup();

// Publish topic: <base>/rpc
_wsPublishTopic := "";
Stu.StrConcatW(pstFrom:=ADR(_wsMqttTopicBase), pstTo:=ADR(_wsPublishTopic), iBufferSize:=GC.STRING_SIZE_TOPIC);
Stu.StrConcatW(pstFrom:=ADR("/rpc"),           pstTo:=ADR(_wsPublishTopic), iBufferSize:=GC.STRING_SIZE_TOPIC);

// Event topic: <base>/events/rpc
_wsMqttTopicEvent := "";
Stu.StrConcatW(pstFrom:=ADR(_wsMqttTopicBase), pstTo:=ADR(_wsMqttTopicEvent), iBufferSize:=GC.STRING_SIZE_TOPIC);
Stu.StrConcatW(pstFrom:=ADR("/events/rpc"),    pstTo:=ADR(_wsMqttTopicEvent), iBufferSize:=GC.STRING_SIZE_TOPIC);

// Status topic: <base>/status/rpc
_wsMqttTopicStatus := "";
Stu.StrConcatW(pstFrom:=ADR(_wsMqttTopicBase), pstTo:=ADR(_wsMqttTopicStatus), iBufferSize:=GC.STRING_SIZE_TOPIC);
Stu.StrConcatW(pstFrom:=ADR("/status/rpc"),    pstTo:=ADR(_wsMqttTopicStatus), iBufferSize:=GC.STRING_SIZE_TOPIC);
END_METHOD

// =============================================================================
// METHOD newMessage
// -----------------------------------------------------------------------------
// Evaluates event and status RPC messages and takes over the generic
// fields (PCB temperature, RSSI, SSID, MAC).
// =============================================================================
METHOD newMessage : BOOL
SUPER^.newMessage();

// Event OR status contain temperature and RSSI.
IF (_fbMqttSubscriber.wsLastTopic = _wsMqttTopicEvent) OR
   (_fbMqttSubscriber.wsLastTopic = _wsMqttTopicStatus) THEN
    fTemperaturePcb := GET_LREAL_FROM_VALUE(fTemperaturePcb, GET_VALUE_FROM_MSG('temperature":{"tC', ADR(_sSubscribedMessage)));
    iRssi           := GET_INT_FROM_VALUE  (iRssi,           GET_VALUE_FROM_MSG('rssi',              ADR(_sSubscribedMessage)));
END_IF

// Only status contains SSID/BSSID.
IF (_fbMqttSubscriber.wsLastTopic = _wsMqttTopicStatus) THEN
    sSsid  := GET_STRING_FROM_VALUE(sSsid,  GET_VALUE_FROM_MSG('ssid',  ADR(_sSubscribedMessage)));
    sMacId := GET_STRING_FROM_VALUE(sMacId, GET_VALUE_FROM_MSG('bssid', ADR(_sSubscribedMessage)));
END_IF
END_METHOD

END_FUNCTION_BLOCK

// xlh_base/app/IoT/DEVICES/IDeviceShelly
// =============================================================================
// IDeviceShelly
// -----------------------------------------------------------------------------
// Marker interface for Shelly devices with native MQTT/JSON-RPC
// (implemented by _200_FB_DEVICE_SHELLY_BASE).
// =============================================================================
INTERFACE IDeviceShelly

END_INTERFACE

// xlh_base/app/IoT/DEVICES/_202_FB_DEVICE_SHELLY_1PM_TEMP
// =============================================================================
// _202_FB_DEVICE_SHELLY_1PM_TEMP
// -----------------------------------------------------------------------------
// Variant of the Shelly Plus 1PM with three external temperature sensors
// (add-on temperature module). Reads the three temperature values from the
// "temperature:100/101/102" properties and calculates their mean value.
//
// Case distinction when parsing:
//   - Event message:  ..."temperature:100":{"tC":21.0,"tF":...}
//   - Status message: ..."temperature:100":{"id":100,"tC":21.0,"tF":...}
// =============================================================================
FUNCTION_BLOCK _202_FB_DEVICE_SHELLY_1PM_TEMP EXTENDS _201_FB_DEVICE_SHELLY_1PM_PLUG
VAR_OUTPUT
    fTemperature1    : LREAL;       // Sensor 100 (°C)
    fTemperature2    : LREAL;       // Sensor 101 (°C)
    fTemperature3    : LREAL;       // Sensor 102 (°C)
    fTemperatureMean : LREAL;       // Mean value of the three sensors (°C)
END_VAR

SUPER^();
fTemperatureMean := (fTemperature1 + fTemperature2 + fTemperature3) / 3.0;

// =============================================================================
// METHOD newMessage
// -----------------------------------------------------------------------------
// Reads the three external temperature sensors. The two different key
// forms (with/without the "id" entry) are tried one after the other; on an
// empty return value, the previous value is kept.
// =============================================================================
METHOD newMessage : BOOL
SUPER^.newMessage();

IF (_fbMqttSubscriber.wsLastTopic = _wsMqttTopicEvent) OR
   (_fbMqttSubscriber.wsLastTopic = _wsMqttTopicStatus) THEN
    fTemperature1 := GET_LREAL_FROM_VALUE(fTemperature1, GET_VALUE_FROM_MSG('temperature:100":{"id": 100,"tC', ADR(_sSubscribedMessage)));
    fTemperature1 := GET_LREAL_FROM_VALUE(fTemperature1, GET_VALUE_FROM_MSG('temperature:100":{"tC',           ADR(_sSubscribedMessage)));
    fTemperature2 := GET_LREAL_FROM_VALUE(fTemperature2, GET_VALUE_FROM_MSG('temperature:101":{"id": 101,"tC', ADR(_sSubscribedMessage)));
    fTemperature2 := GET_LREAL_FROM_VALUE(fTemperature2, GET_VALUE_FROM_MSG('temperature:101":{"tC',           ADR(_sSubscribedMessage)));
    fTemperature3 := GET_LREAL_FROM_VALUE(fTemperature3, GET_VALUE_FROM_MSG('temperature:102":{"id": 102,"tC', ADR(_sSubscribedMessage)));
    fTemperature3 := GET_LREAL_FROM_VALUE(fTemperature3, GET_VALUE_FROM_MSG('temperature:102":{"tC',           ADR(_sSubscribedMessage)));
END_IF
END_METHOD

END_FUNCTION_BLOCK

// xlh_base/app/IoT/DEVICES/_201_FB_DEVICE_SHELLY_1PM_PLUG
// =============================================================================
// _201_FB_DEVICE_SHELLY_1PM_PLUG
// -----------------------------------------------------------------------------
// FB for a Shelly Plus 1PM (plug with energy metering).
//
// Functionality:
//   - Receives measurement/switching state via the Shelly event/status RPC
//     topic.
//   - Switches the relay via Switch.Set (publish on <base>/rpc).
//   - Calculates its own cumulative energy balance (fElectricalEnergy) by
//     integrating the measured active power. bResetEnergy resets the
//     counter.
//
// Trigger logic for the relay set command:
//   A publish is made when (a) the request changes (R/F trigger) or (b) the
//   request differs from the reported relay state for longer than
//   _tACTION_TIME_NOT_EQUAL (repeat for synchronization).
// =============================================================================
FUNCTION_BLOCK _201_FB_DEVICE_SHELLY_1PM_PLUG EXTENDS _200_FB_DEVICE_SHELLY_BASE
VAR_INPUT
    bRelais       : BOOL;       // Requested state of the relay
    bResetEnergy  : BOOL;       // TRUE -> reset the integrated energy counter
END_VAR
VAR_OUTPUT
    bRelaisState        : BOOL;     // Actual state of the relay (reported by the device)
    fVoltage            : LREAL;    // Mains voltage (V)
    fCurrent            : LREAL;    // Current (A)
    fPower              : LREAL;    // Active power (W)
    fElectricalEnergy   : LREAL;    // Integrated electrical energy (W·s)
END_VAR
VAR
    _fbRtRelais             : R_TRIG;   // Rising edge of the request
    _fbFtRelais             : F_TRIG;   // Falling edge of the request
    _fbTonDiffRelaisState   : TON;      // Watchdog: request <> state for longer than _tACTION_TIME_NOT_EQUAL
END_VAR
VAR CONSTANT
    _tACTION_TIME_NOT_EQUAL : TIME := T#500MS; // Time after which a sync publish is forced
END_VAR

SUPER^();

// Own energy metering (integration over the cycle time).
IF bResetEnergy THEN
    fElectricalEnergy := 0.0;
ELSE
    fElectricalEnergy := fElectricalEnergy + fPower * TASK_INFO.fCycleTime;
END_IF

// =============================================================================
// METHOD publisher
// -----------------------------------------------------------------------------
// Sends a Switch.Set RPC command when required to track the relay state.
// The SUPER implementation takes care of the actual send processing of
// the queue.
// =============================================================================
METHOD publisher : BOOL
VAR
    bPublish        : BOOL;
    sPublishMessage : STRING(GC.STRING_SIZE_MESSAGE_TX);
END_VAR

// Combine the trigger conditions.
THIS^._fbTonDiffRelaisState(IN := ((THIS^.bRelais <> THIS^.bRelaisState) AND NOT _fbTonDiffRelaisState.Q),
                            PT := THIS^._tACTION_TIME_NOT_EQUAL);
THIS^._fbRtRelais(CLK := THIS^.bRelais);
THIS^._fbFtRelais(CLK := THIS^.bRelais);
bPublish := _fbTonDiffRelaisState.Q OR _fbRtRelais.Q OR _fbFtRelais.Q;

IF bPublish THEN
    // {"id":1, "src":"<base>/relais", "method":"Switch.Set", "params":{"id":0, "on":true|false}}
    sPublishMessage := '{"id":1, "src":"';
    Stu.StrConcatA(pstFrom:=ADR(THIS^.sMqttTopicBase),
                   pstTo  :=ADR(sPublishMessage),
                   iBufferSize:=GC.STRING_SIZE_MESSAGE_TX);
    Stu.StrConcatA(pstFrom:=ADR('/relais", "method":"Switch.Set", "params":{"id":0, "on":'),
                   pstTo  :=ADR(sPublishMessage),
                   iBufferSize:=GC.STRING_SIZE_MESSAGE_TX);
    IF THIS^.bRelais THEN
        Stu.StrConcatA(pstFrom:=ADR('true}}'),  pstTo:=ADR(sPublishMessage), iBufferSize:=GC.STRING_SIZE_MESSAGE_TX);
    ELSE
        Stu.StrConcatA(pstFrom:=ADR('false}}'), pstTo:=ADR(sPublishMessage), iBufferSize:=GC.STRING_SIZE_MESSAGE_TX);
    END_IF
    THIS^.pushFifoPublish(THIS^._wsPublishTopic, sPublishMessage);
END_IF

SUPER^.publisher();
END_METHOD

// =============================================================================
// METHOD newMessage
// -----------------------------------------------------------------------------
// Reads the switching state and the measurements from event/status RPC
// responses. An example status message is attached at the end of the
// method code.
// =============================================================================
METHOD newMessage : BOOL
SUPER^.newMessage();

IF (_fbMqttSubscriber.wsLastTopic = _wsMqttTopicEvent) OR
   (_fbMqttSubscriber.wsLastTopic = _wsMqttTopicStatus) THEN
    bRelaisState := GET_BOOL_FROM_VALUE (bRelaisState, GET_VALUE_FROM_MSG('output',  ADR(_sSubscribedMessage)));
    fVoltage     := GET_LREAL_FROM_VALUE(fVoltage,     GET_VALUE_FROM_MSG('voltage', ADR(_sSubscribedMessage)));
    fCurrent     := GET_LREAL_FROM_VALUE(fCurrent,     GET_VALUE_FROM_MSG('current', ADR(_sSubscribedMessage)));
    fPower       := GET_LREAL_FROM_VALUE(fPower,       GET_VALUE_FROM_MSG('apower',  ADR(_sSubscribedMessage)));
END_IF

(*
// FixMe: total energy from status Message

Topic: shellyplus1pm-51/status/rpc QoS: 0
{"id":1,"src":"shellyplus1pm-...","dst":"shellyplus1pm-51/status",
 "result":{"ble":{},"cloud":{"connected":false},
   "input:0":{"id":0,"state":false},"mqtt":{"connected":true},
   "switch:0":{"id":0, "source":"MQTT", "output":false, "apower":0.0,
               "voltage":236.0, "current":0.000,
               "aenergy":{"total":2431.000, "by_minute":[0,0,0],
                          "minute_ts":1765258740},
               "temperature":{"tC":38.2, "tF":100.8}},
   "sys":{"mac":"...", "uptime":380, ...},
   "wifi":{"sta_ip":"...", "ssid":"...", "bssid":"...", "rssi":-28},
   "ws":{"connected":false}}}
*)
END_METHOD

END_FUNCTION_BLOCK

